PROPERTY PUBLIC Busy : BOOL
GET
Busy := asyncResponse <> 0;
END_GET
END_PROPERTY

METHOD PUBLIC CyclicCall
VAR_INPUT
END_VAR
timer(in := Busy, pt := T#1S);

IF timer.Q THEN
	asyncResponse.CompleteWithString(result);
	asyncResponse := 0;
	result := '';
END_IF
END_METHOD

METHOD Handle
VAR_INPUT
	Parameters : I_Deserializer;
	Response : I_SynchronousRpcResponse;
END_VAR
VAR
	deserializerFeedback : DeserializerFeedback;
	echo : T_MAXSTRING;
END_VAR
IF Busy THEN
	Response.RejectWithError('HANDLER_TOO_BUSY','Already processing response');
	RETURN;
END_IF

IF NOT Parameters.TryGetKeyString('Echo', echo, deserializerFeedback) THEN
	Response.RejectWithError('MISSING_PARAMETER','Missing Echo parameter');
	RETURN;
END_IF

result := echo;
Response.TryMakeAsynchronous(asyncResponse);
END_METHOD

END_FUNCTION_BLOCK

// ---- mobject-server/Mocks/RejectWithMessageAsyncHandler.TcPOU
FUNCTION_BLOCK RejectWithMessageAsyncHandler IMPLEMENTS I_AsynchronousRpcHandler
VAR
END_VAR

METHOD Handle
VAR_INPUT
	Parameters : I_Deserializer;
	Response : I_AsynchronousRpcResponse;
END_VAR
VAR
END_VAR
Response.RejectWithError('EXAMPLE_ERROR_CODE','This is the reject message');
END_METHOD

END_FUNCTION_BLOCK

// ---- mobject-server/Mocks/RejectWithMessageSyncHandler.TcPOU
FUNCTION_BLOCK RejectWithMessageSyncHandler IMPLEMENTS I_SynchronousRpcHandler
VAR
END_VAR

METHOD Handle
VAR_INPUT
	Parameters : I_Deserializer;
	Response : I_SynchronousRpcResponse;
END_VAR
VAR
END_VAR
Response.RejectWithError('EXAMPLE_ERROR_CODE','This is the reject message');
END_METHOD

END_FUNCTION_BLOCK

// ---- mobject-server/_Internal/ChunkedRequestData_TestSuite.TcPOU
FUNCTION_BLOCK ChunkedRequestData_TestSuite EXTENDS TcUnit.FB_TestSuite
VAR
END_VAR

TestChunkedPayloadStoredCorrectly_10Chunks();
TestChunkedPayloadStoredCorrectly_2Chunks();
TestCorrectPayloadSizeInBytes_20Bytes();
TestCorrectPayloadSizeInBytes_100Bytes();
TestIsCompleteOnceAllChunksAdded();
TestTryAddChunkedPayloadReturnsFalseWhenTooBig();
TestTryAddChunkedPayloadReturnsTrueWhenValid();
TestTryAddChunkedPayloadRejectsOutOfOrderChunk();
TestTryAddChunkedPayloadRejectsDuplicateChunk();

METHOD TestChunkedPayloadStoredCorrectly_10Chunks
VAR
	chunkedRequestData : ChunkedRequestData(3,10); // results in 30 bytes
	dataChunk1 : STRING(2) := 'ab'; // results in 3 bytes
	dataChunk2 : STRING(2) := 'cd'; // results in 3 bytes
	dataChunk3 : STRING(2) := 'ef'; // results in 3 bytes
	dataChunk4 : STRING(2) := 'gh'; // results in 3 bytes
	dataChunk5 : STRING(2) := 'ij'; // results in 3 bytes
	dataChunk6 : STRING(2) := 'kl'; // results in 3 bytes
	dataChunk7 : STRING(2) := 'mn'; // results in 3 bytes
	dataChunk8 : STRING(2) := 'op'; // results in 3 bytes
	dataChunk9 : STRING(2) := 'qr'; // results in 3 bytes
	dataChunk10 : STRING(2) := 'st'; // results in 3 bytes
	dataAddress : PVOID;
	dataSize : UDINT;
	result : STRING(29);
	expected : STRING(29) := 'abcdefghijklmnopqrst'; // results in 30 bytes
END_VAR
TEST('TestChunkedPayloadStoredCorrectly_10Chunks');

memset(ADR(result),0,SIZEOF(result));

chunkedRequestData.TryAddChunkedPayload(ADR(dataChunk1), SIZEOF(dataChunk1), 1);
chunkedRequestData.TryAddChunkedPayload(ADR(dataChunk2), SIZEOF(dataChunk2), 2);
chunkedRequestData.TryAddChunkedPayload(ADR(dataChunk3), SIZEOF(dataChunk3), 3);
chunkedRequestData.TryAddChunkedPayload(ADR(dataChunk4), SIZEOF(dataChunk4), 4);
chunkedRequestData.TryAddChunkedPayload(ADR(dataChunk5), SIZEOF(dataChunk5), 5);
chunkedRequestData.TryAddChunkedPayload(ADR(dataChunk6), SIZEOF(dataChunk6), 6);
chunkedRequestData.TryAddChunkedPayload(ADR(dataChunk7), SIZEOF(dataChunk7), 7);
chunkedRequestData.TryAddChunkedPayload(ADR(dataChunk8), SIZEOF(dataChunk8), 8);
chunkedRequestData.TryAddChunkedPayload(ADR(dataChunk9), SIZEOF(dataChunk9), 9);
chunkedRequestData.TryAddChunkedPayload(ADR(dataChunk10), SIZEOF(dataChunk10), 10);

dataAddress := chunkedRequestData.PayloadAddress;
dataSize := chunkedRequestData.PayloadSizeInBytes;

memcpy(ADR(result),dataAddress,dataSize);

AssertEquals(
	Expected := expected,
	Actual := result,
	Message := 'Did not correctly assemble the chunked string data'
);

TEST_FINISHED();
END_METHOD

METHOD TestChunkedPayloadStoredCorrectly_2Chunks
VAR
	chunkedRequestData : ChunkedRequestData(4,2); // results in 8 bytes
	dataChunk1 : STRING(3) := 'foo'; // results in 4 bytes
	dataChunk2 : STRING(3) := 'bar'; // results in 4 bytes
	dataAddress : PVOID;
	dataSize : UDINT;
	result : STRING(7);
	expected : STRING(7) := 'foobar'; // results in 8 bytes
END_VAR
TEST('TestChunkedPayloadStoredCorrectly_2Chunks');

memset(ADR(result),0,SIZEOF(result));

chunkedRequestData.TryAddChunkedPayload(ADR(dataChunk1), SIZEOF(dataChunk1), 1);
chunkedRequestData.TryAddChunkedPayload(ADR(dataChunk2), SIZEOF(dataChunk2), 2);

dataAddress := chunkedRequestData.PayloadAddress;
dataSize := chunkedRequestData.PayloadSizeInBytes;

memcpy(ADR(result),dataAddress,dataSize);

AssertEquals(
	Expected := expected,
	Actual := result,
	Message := 'Did not correctly assemble the chunked string data'
);

TEST_FINISHED();
END_METHOD

METHOD TestCorrectPayloadSizeInBytes_100Bytes
VAR
	chunkedRequestData : ChunkedRequestData(20,5);
	result : UDINT;
	expected : UDINT := 100;
END_VAR
TEST('TestCorrectPayloadSizeInBytes_100Bytes');

result := chunkedRequestData.PayloadSizeInBytes;

AssertEquals(
	Expected := expected,
	Actual := result,
	Message := 'Did not create the correct payload size based on the constructor arguments'
);

TEST_FINISHED();
END_METHOD

METHOD TestCorrectPayloadSizeInBytes_20Bytes
VAR
	chunkedRequestData : ChunkedRequestData(2,10);
	result : UDINT;
	expected : UDINT := 20;
END_VAR
TEST('TestCorrectPayloadSizeInBytes_20Bytes');

result := chunkedRequestData.PayloadSizeInBytes;

AssertEquals(
	Expected := expected,
	Actual := result,
	Message := 'Did not create the correct payload size based on the constructor arguments'
);

TEST_FINISHED();
END_METHOD

METHOD TestIsCompleteOnceAllChunksAdded
VAR
	chunkedRequestData : ChunkedRequestData(4,2);
	dataChunk1 : STRING(3) := 'foo';
	dataChunk2 : STRING(3) := 'bar';
	isComplete : BOOL;
END_VAR
TEST('TestIsCompleteOnceAllChunksAdded');

isComplete := chunkedRequestData.IsComplete;

AssertFalse(
	Condition := isComplete,
	Message := 'Incorrectly reported as IsComplete with 0/2 chunks added'
);

chunkedRequestData.TryAddChunkedPayload(ADR(dataChunk1), SIZEOF(dataChunk1), 1);
isComplete := chunkedRequestData.IsComplete;

AssertFalse(
	Condition := isComplete,
	Message := 'Incorrectly reported as IsComplete with 1/2 chunks added'
);

chunkedRequestData.TryAddChunkedPayload(ADR(dataChunk2), SIZEOF(dataChunk2), 2);
isComplete := chunkedRequestData.IsComplete;

AssertTrue(
	Condition := isComplete,
	Message := 'Failed to reported IsComplete with 2/2 chunks added'
);

TEST_FINISHED();
END_METHOD

METHOD TestTryAddChunkedPayloadReturnsFalseWhenTooBig
VAR
	chunkedRequestData : ChunkedRequestData(4,1);
	dataChunk : STRING(10) := 'foo';
	added : BOOL;
END_VAR
TEST('TestTryAddChunkedPayloadReturnsFalseWhenTooBig');

added := chunkedRequestData.TryAddChunkedPayload(ADR(dataChunk), SIZEOF(dataChunk), 1);

AssertFalse(
	Condition := added,
	Message := 'Incorrectly reported that the try was successful'
);

TEST_FINISHED();
END_METHOD

METHOD TestTryAddChunkedPayloadRejectsOutOfOrderChunk
VAR
	chunkedRequestData : ChunkedRequestData(4,3);
	dataChunk : STRING(3) := 'foo';
	added : BOOL;
END_VAR
TEST('TestTryAddChunkedPayloadRejectsOutOfOrderChunk');

// chunk 2 arriving before chunk 1 cannot be appended in the right place
added := chunkedRequestData.TryAddChunkedPayload(ADR(dataChunk), SIZEOF(dataChunk), 2);

AssertFalse(
	Condition := added,
	Message := 'A chunk which is not the one due next must be rejected, not appended out of order'
);

TEST_FINISHED();
END_METHOD

METHOD TestTryAddChunkedPayloadRejectsDuplicateChunk
VAR
	chunkedRequestData : ChunkedRequestData(4,3);
	dataChunk : STRING(3) := 'foo';
	firstAdd : BOOL;
	duplicateAdd : BOOL;
END_VAR
TEST('TestTryAddChunkedPayloadRejectsDuplicateChunk');

firstAdd := chunkedRequestData.TryAddChunkedPayload(ADR(dataChunk), SIZEOF(dataChunk), 1);
duplicateAdd := chunkedRequestData.TryAddChunkedPayload(ADR(dataChunk), SIZEOF(dataChunk), 1);

AssertTrue(
	Condition := firstAdd,
	Message := 'The first chunk should have been accepted'
);

// resending chunk 1 would otherwise append it twice and count twice towards completion
AssertFalse(
	Condition := duplicateAdd,
	Message := 'A repeated chunk must be rejected rather than appended a second time'
);

TEST_FINISHED();
END_METHOD

METHOD TestTryAddChunkedPayloadReturnsTrueWhenValid
VAR
	chunkedRequestData : ChunkedRequestData(4,1);
	dataChunk : STRING(3) := 'foo';
	added : BOOL;
END_VAR
TEST('TestTryAddChunkedPayloadReturnsTrueWhenValid');

added := chunkedRequestData.TryAddChunkedPayload(ADR(dataChunk), SIZEOF(dataChunk), 1);

AssertTrue(
	Condition := added,
	Message := 'Incorrectly reported that the try failed'
);

TEST_FINISHED();
END_METHOD

END_FUNCTION_BLOCK

// ---- mobject-server/_Internal/AsyncResponseSessionData_TestSuite.TcPOU
FUNCTION_BLOCK AsyncResponseSessionData_TestSuite EXTENDS TcUnit.FB_TestSuite
VAR
END_VAR

TestNewResponseIsPending();
TestFreshResponseHasNotExpired();
TestZeroMaxAgeDisablesTheDeadline();
TestCompletedResponseIsNoLongerPending();
TestRejectedResponseIsNoLongerPending();

METHOD TestCompletedResponseIsNoLongerPending
VAR
	asyncResponseSessionData : AsyncResponseSessionData(SuggestedRetryDelayInMs := 0, MaxAge := T#60S);
END_VAR
TEST('TestCompletedResponseIsNoLongerPending');

asyncResponseSessionData.Success();

AssertFalse(
	Condition := asyncResponseSessionData.IsPending,
	Message := 'A response which has completed should no longer report as pending'
);

TEST_FINISHED();
END_METHOD

METHOD TestFreshResponseHasNotExpired
VAR
	asyncResponseSessionData : AsyncResponseSessionData(SuggestedRetryDelayInMs := 0, MaxAge := T#60S);
END_VAR
TEST('TestFreshResponseHasNotExpired');

AssertFalse(
	Condition := asyncResponseSessionData.HasExpired,
	Message := 'A response created this cycle cannot already be past a 60s deadline'
);

TEST_FINISHED();
END_METHOD

METHOD TestNewResponseIsPending
VAR
	asyncResponseSessionData : AsyncResponseSessionData(SuggestedRetryDelayInMs := 0, MaxAge := T#60S);
END_VAR
TEST('TestNewResponseIsPending');

AssertTrue(
	Condition := asyncResponseSessionData.IsPending,
	Message := 'A newly created response should be pending until the handler completes it'
);

TEST_FINISHED();
END_METHOD

METHOD TestRejectedResponseIsNoLongerPending
VAR
	asyncResponseSessionData : AsyncResponseSessionData(SuggestedRetryDelayInMs := 0, MaxAge := T#60S);
END_VAR
TEST('TestRejectedResponseIsNoLongerPending');

asyncResponseSessionData.Error('SOME_CODE', 'some message');

AssertFalse(
	Condition := asyncResponseSessionData.IsPending,
	Message := 'A response which has been rejected should no longer report as pending'
);

TEST_FINISHED();
END_METHOD

METHOD TestZeroMaxAgeDisablesTheDeadline
VAR
	asyncResponseSessionData : AsyncResponseSessionData(SuggestedRetryDelayInMs := 0, MaxAge := T#0S);
END_VAR
TEST('TestZeroMaxAgeDisablesTheDeadline');

// T#0S is the documented way to switch the deadline off.  It must not be read
// as 'expires immediately', which would fail every asynchronous call.
AssertFalse(
	Condition := asyncResponseSessionData.HasExpired,
	Message := 'A max age of T#0S should disable the deadline, not expire instantly'
);

TEST_FINISHED();
END_METHOD

END_FUNCTION_BLOCK

// ---- mobject-server/Mocks/AdjustableSizeReplyRpcHandler.TcPOU
FUNCTION_BLOCK AdjustableSizeReplyRpcHandler IMPLEMENTS I_SynchronousRpcHandler
VAR
END_VAR

METHOD Handle
VAR_INPUT
	Parameters : I_Deserializer;
	Response : I_SynchronousRpcResponse;
END_VAR
VAR
	deserializerFeedback : DeserializerFeedback;
	size : UDINT;
	pBytes : POINTER TO BYTE;
	currentPos : POINTER TO BYTE;
	i : UDINT;
	count : BYTE;
END_VAR
IF NOT Parameters.TryGetKeyUdint('Size', size, deserializerFeedback) THEN
	Response.RejectWithError('MISSING_PARAMETER','Missing Size parameter');
	RETURN;
END_IF

IF size = 0 THEN 
	Response.CompleteWithNull();
END_IF

pBytes := __NEW(BYTE, size);
FOR i := 0 TO size -1 DO
	currentPos := pBytes + i;
	currentPos^ := count;
	count := count + 1;
END_FOR

Response.CompleteWithBytesAsHex(pBytes, UDINT_TO_DINT(size));

__Delete(pBytes);
END_METHOD

END_FUNCTION_BLOCK

// ---- mobject-collections/MobjectCollectionsExample.TcPOU
PROGRAM MobjectCollectionsExample
VAR
END_VAR

END_PROGRAM

// ---- mobject-collections/Tests/Mocks/EventHandlers/CollectionEventHandlerBase.TcPOU
FUNCTION_BLOCK ABSTRACT CollectionEventHandlerBase IMPLEMENTS I_EventHandler
VAR
	_eventReceived : BOOL;
	fromExpected : BOOL;
END_VAR

PROPERTY PUBLIC EventReceived : BOOL
GET // PUBLIC
EventReceived := _eventReceived;
END_GET
END_PROPERTY

PROPERTY PUBLIC FromExpectedOriginator : BOOL
GET // PUBLIC
FromExpectedOriginator := fromExpected;
END_GET
END_PROPERTY

METHOD PUBLIC ABSTRACT HandleEvent
VAR_INPUT
	Event : I_Event;
END_VAR
END_METHOD

METHOD PUBLIC Reset
_eventReceived := FALSE;
fromExpected := FALSE;
END_METHOD

END_FUNCTION_BLOCK

// ---- mobject-collections/Tests/Mocks/EventHandlers/KeyValueCollectionDisposedEventHandler.TcPOU
FUNCTION_BLOCK KeyValueCollectionDisposedEventHandler EXTENDS KeyValueCollectionEventHandler

METHOD PUBLIC HandleEvent
VAR_INPUT
	Event : I_Event;
END_VAR
VAR
	disposedEvent : I_KeyValueCollectionDisposedEvent;
END_VAR
IF __QUERYINTERFACE(Event, disposedEvent) THEN
	_eventReceived := TRUE;
	fromExpected := disposedEvent.Target = expectedOriginator;
END_IF
END_METHOD

END_FUNCTION_BLOCK

// ---- mobject-collections/Tests/Mocks/EventHandlers/KeyValueCollectionEventHandler.TcPOU
FUNCTION_BLOCK ABSTRACT KeyValueCollectionEventHandler EXTENDS CollectionEventHandlerBase
VAR
	expectedOriginator : I_KeyValueCollection;
END_VAR

METHOD FB_init : BOOL
VAR_INPUT
	bInitRetains : BOOL; // if TRUE, the retain variables are initialized (warm start / cold start)
	bInCopyCode : BOOL;  // if TRUE, the instance afterwards gets moved into the copy code (online change)
	ExpectedOriginator : I_KeyValueCollection;
END_VAR
SetExpectedOriginator(ExpectedOriginator);
END_METHOD

METHOD PUBLIC SetExpectedOriginator
VAR_INPUT
	ExpectedOriginator : I_KeyValueCollection;
END_VAR
THIS^.expectedOriginator := ExpectedOriginator;
END_METHOD

END_FUNCTION_BLOCK

// ---- mobject-converters/Tests/BYTE_TO_TestSuite.TcPOU
FUNCTION_BLOCK PUBLIC BYTE_TO_TestSuite EXTENDS TcUnit.FB_TestSuite
VAR
END_VAR

Check_BYTE_TO_BOOL_Max();
Check_BYTE_TO_BOOL_Min();
Check_BYTE_TO_BYTE_Max();
Check_BYTE_TO_BYTE_Min();
Check_BYTE_TO_WORD_Max();
Check_BYTE_TO_WORD_Min();
Check_BYTE_TO_DWORD_Max();
Check_BYTE_TO_DWORD_Min();
Check_BYTE_TO_LWORD_Max();
Check_BYTE_TO_LWORD_Min();
Check_BYTE_TO_SINT_Max();
Check_BYTE_TO_SINT_Min();
Check_BYTE_TO_SINT_TooHigh();
Check_BYTE_TO_INT_Max();
Check_BYTE_TO_INT_Min();
Check_BYTE_TO_DINT_Max();
Check_BYTE_TO_DINT_Min();
Check_BYTE_TO_LINT_Max();
Check_BYTE_TO_LINT_Min();
Check_BYTE_TO_USINT_Max();
Check_BYTE_TO_USINT_Min();
Check_BYTE_TO_UINT_Max();
Check_BYTE_TO_UINT_Min();
Check_BYTE_TO_UDINT_Max();
Check_BYTE_TO_UDINT_Min();
Check_BYTE_TO_ULINT_Max();
Check_BYTE_TO_ULINT_Min();
Check_BYTE_TO_REAL_Max();
Check_BYTE_TO_REAL_Min();
Check_BYTE_TO_LREAL_Max();
Check_BYTE_TO_LREAL_Min();
Check_BYTE_TO_TIME_Max();
Check_BYTE_TO_TIME_Min();
Check_BYTE_TO_TOD_Max();
Check_BYTE_TO_TOD_Min();
Check_BYTE_TO_DATE_Max();
Check_BYTE_TO_DATE_Min();
Check_BYTE_TO_DT_Max();
Check_BYTE_TO_DT_Min();
Check_BYTE_TO_STRING_Max();
Check_BYTE_TO_STRING_Min();

METHOD PUBLIC Check_BYTE_TO_BOOL_Max
VAR
	value : BYTE := DatatypeLimits.BYTE_MAX_VALUE;
	actual : BOOL;
	converted : BOOL;
	equal : BOOL;
END_VAR
TEST('Check_BYTE_TO_BOOL_Max');

// @TEST-RUN
converted := TryConvert_BYTE_TO_Destination(value, actual);
equal := actual = BYTE_TO_BOOL(value);

// @TEST-ASSERT
AssertTrue(Condition := equal, Message := 'Did not convert BYTE to BOOL correctly');
AssertTrue(Condition := converted, Message := 'Did not report BYTE to BOOL conversion was successful');

TEST_FINISHED();
END_METHOD

METHOD PUBLIC Check_BYTE_TO_BOOL_Min
VAR
	value : BYTE := DatatypeLimits.BYTE_MIN_VALUE;
	actual : BOOL;
	converted : BOOL;
	equal : BOOL;
END_VAR
TEST('Check_BYTE_TO_BOOL_Min');

// @TEST-RUN
converted := TryConvert_BYTE_TO_Destination(value, actual);
equal := actual = BYTE_TO_BOOL(value);

// @TEST-ASSERT
AssertTrue(Condition := equal, Message := 'Did not convert BYTE to BOOL correctly');
AssertTrue(Condition := converted, Message := 'Did not report BYTE to BOOL conversion was successful');

TEST_FINISHED();
END_METHOD

METHOD PUBLIC Check_BYTE_TO_BYTE_Max
VAR
	value : BYTE := DatatypeLimits.BYTE_MAX_VALUE;
	actual : BYTE;
	converted : BOOL;
	equal : BOOL;
END_VAR
TEST('Check_BYTE_TO_BYTE_Max');

// @TEST-RUN
converted := TryConvert_BYTE_TO_Destination(value, actual);
equal := actual = value;

// @TEST-ASSERT
AssertTrue(Condition := equal, Message := 'Did not convert BYTE to BYTE correctly');
AssertTrue(Condition := converted, Message := 'Did not report BYTE to BYTE conversion was successful');

TEST_FINISHED();
END_METHOD

METHOD PUBLIC Check_BYTE_TO_BYTE_Min
VAR
	value : BYTE := DatatypeLimits.BYTE_MIN_VALUE;
	actual : BYTE;
	converted : BOOL;
	equal : BOOL;
END_VAR
TEST('Check_BYTE_TO_BYTE_Min');

// @TEST-RUN
converted := TryConvert_BYTE_TO_Destination(value, actual);
equal := actual = value;

// @TEST-ASSERT
AssertTrue(Condition := equal, Message := 'Did not convert BYTE to BYTE correctly');
AssertTrue(Condition := converted, Message := 'Did not report BYTE to BYTE conversion was successful');

TEST_FINISHED();
END_METHOD

METHOD PUBLIC Check_BYTE_TO_DATE_Max
VAR
	value : BYTE := DatatypeLimits.BYTE_MAX_VALUE;
	actual : DATE;
	converted : BOOL;
	equal : BOOL;
END_VAR
TEST('Check_BYTE_TO_DATE_Max');

// @TEST-RUN
converted := TryConvert_BYTE_TO_Destination(value, actual);
equal := actual = BYTE_TO_DATE(value);

// @TEST-ASSERT
AssertTrue(Condition := equal, Message := 'Did not convert BYTE to DATE correctly');
AssertTrue(Condition := converted, Message := 'Did not report BYTE to DATE conversion was successful');

TEST_FINISHED();
END_METHOD

METHOD PUBLIC Check_BYTE_TO_DATE_Min
VAR
	value : BYTE := DatatypeLimits.BYTE_MIN_VALUE;
	actual : DATE;
	converted : BOOL;
	equal : BOOL;
END_VAR
TEST('Check_BYTE_TO_DATE_Min');

// @TEST-RUN
converted := TryConvert_BYTE_TO_Destination(value, actual);
equal := actual = BYTE_TO_DATE(value);

// @TEST-ASSERT
AssertTrue(Condition := equal, Message := 'Did not convert BYTE to DATE correctly');
AssertTrue(Condition := converted, Message := 'Did not report BYTE to DATE conversion was successful');

TEST_FINISHED();
END_METHOD

METHOD PUBLIC Check_BYTE_TO_DINT_Max
VAR
	value : BYTE := DatatypeLimits.BYTE_MAX_VALUE;
	actual : DINT;
	converted : BOOL;
	equal : BOOL;
END_VAR
TEST('Check_BYTE_TO_DINT_Max');

// @TEST-RUN
converted := TryConvert_BYTE_TO_Destination(value, actual);
equal := actual = BYTE_TO_DINT(value);

// @TEST-ASSERT
AssertTrue(Condition := equal, Message := 'Did not convert BYTE to DINT correctly');
AssertTrue(Condition := converted, Message := 'Did not report BYTE to DINT conversion was successful');

TEST_FINISHED();
END_METHOD

METHOD PUBLIC Check_BYTE_TO_DINT_Min
VAR
	value : BYTE := DatatypeLimits.BYTE_MIN_VALUE;
	actual : DINT;
	converted : BOOL;
	equal : BOOL;
END_VAR
TEST('Check_BYTE_TO_DINT_Min');

// @TEST-RUN
converted := TryConvert_BYTE_TO_Destination(value, actual);
equal := actual = BYTE_TO_DINT(value);

// @TEST-ASSERT
AssertTrue(Condition := equal, Message := 'Did not convert BYTE to DINT correctly');
AssertTrue(Condition := converted, Message := 'Did not report BYTE to DINT conversion was successful');

TEST_FINISHED();
END_METHOD

METHOD PUBLIC Check_BYTE_TO_DT_Max
VAR
	value : BYTE := DatatypeLimits.BYTE_MAX_VALUE;
	actual : DT;
	converted : BOOL;
	equal : BOOL;
END_VAR
TEST('Check_BYTE_TO_DT_Max');

// @TEST-RUN
converted := TryConvert_BYTE_TO_Destination(value, actual);
equal := actual = BYTE_TO_DT(value);

// @TEST-ASSERT
AssertTrue(Condition := equal, Message := 'Did not convert BYTE to DT correctly');
AssertTrue(Condition := converted, Message := 'Did not report BYTE to DT conversion was successful');

TEST_FINISHED();
END_METHOD

METHOD PUBLIC Check_BYTE_TO_DT_Min
VAR
	value : BYTE := DatatypeLimits.BYTE_MIN_VALUE;
	actual : DT;
	converted : BOOL;
	equal : BOOL;
END_VAR
TEST('Check_BYTE_TO_DT_Min');

// @TEST-RUN
converted := TryConvert_BYTE_TO_Destination(value, actual);
equal := actual = BYTE_TO_DT(value);

// @TEST-ASSERT
AssertTrue(Condition := equal, Message := 'Did not convert BYTE to DT correctly');
AssertTrue(Condition := converted, Message := 'Did not report BYTE to DT conversion was successful');

TEST_FINISHED();
END_METHOD

METHOD PUBLIC Check_BYTE_TO_DWORD_Max
VAR
	value : BYTE := DatatypeLimits.BYTE_MAX_VALUE;
	actual : DWORD;
	converted : BOOL;
	equal : BOOL;
END_VAR
TEST('Check_BYTE_TO_DWORD_Max');

// @TEST-RUN
converted := TryConvert_BYTE_TO_Destination(value, actual);
equal := actual = BYTE_TO_DWORD(value);

// @TEST-ASSERT
AssertTrue(Condition := equal, Message := 'Did not convert BYTE to DWORD correctly');
AssertTrue(Condition := converted, Message := 'Did not report BYTE to DWORD conversion was successful');

TEST_FINISHED();
END_METHOD

METHOD PUBLIC Check_BYTE_TO_DWORD_Min
VAR
	value : BYTE := DatatypeLimits.BYTE_MIN_VALUE;
	actual : DWORD;
	converted : BOOL;
	equal : BOOL;
END_VAR
TEST('Check_BYTE_TO_DWORD_Min');

// @TEST-RUN
converted := TryConvert_BYTE_TO_Destination(value, actual);
equal := actual = BYTE_TO_DWORD(value);

// @TEST-ASSERT
AssertTrue(Condition := equal, Message := 'Did not convert BYTE to DWORD correctly');
AssertTrue(Condition := converted, Message := 'Did not report BYTE to DWORD conversion was successful');

TEST_FINISHED();
END_METHOD

METHOD PUBLIC Check_BYTE_TO_INT_Max
VAR
	value : BYTE := DatatypeLimits.BYTE_MAX_VALUE;
	actual : INT;
	converted : BOOL;
	equal : BOOL;
END_VAR
TEST('Check_BYTE_TO_INT_Max');

// @TEST-RUN
converted := TryConvert_BYTE_TO_Destination(value, actual);
equal := actual = BYTE_TO_INT(value);

// @TEST-ASSERT
AssertTrue(Condition := equal, Message := 'Did not convert BYTE to INT correctly');
AssertTrue(Condition := converted, Message := 'Did not report BYTE to INT conversion was successful');

TEST_FINISHED();
END_METHOD

METHOD PUBLIC Check_BYTE_TO_INT_Min
VAR
	value : BYTE := DatatypeLimits.BYTE_MIN_VALUE;
	actual : INT;
	converted : BOOL;
	equal : BOOL;
END_VAR
TEST('Check_BYTE_TO_INT_Min');

// @TEST-RUN
converted := TryConvert_BYTE_TO_Destination(value, actual);
equal := actual = BYTE_TO_INT(value);

// @TEST-ASSERT
AssertTrue(Condition := equal, Message := 'Did not convert BYTE to INT correctly');
AssertTrue(Condition := converted, Message := 'Did not report BYTE to INT conversion was successful');

TEST_FINISHED();
END_METHOD

METHOD PUBLIC Check_BYTE_TO_LINT_Max
VAR
	value : BYTE := DatatypeLimits.BYTE_MAX_VALUE;
	actual : LINT;
	converted : BOOL;
	equal : BOOL;
END_VAR
TEST('Check_BYTE_TO_LINT_Max');

// @TEST-RUN
converted := TryConvert_BYTE_TO_Destination(value, actual);
equal := actual = BYTE_TO_LINT(value);

// @TEST-ASSERT
AssertTrue(Condition := equal, Message := 'Did not convert BYTE to LINT correctly');
AssertTrue(Condition := converted, Message := 'Did not report BYTE to LINT conversion was successful');

TEST_FINISHED();
END_METHOD

METHOD PUBLIC Check_BYTE_TO_LINT_Min
VAR
	value : BYTE := DatatypeLimits.BYTE_MIN_VALUE;
	actual : LINT;
	converted : BOOL;
	equal : BOOL;
END_VAR
TEST('Check_BYTE_TO_LINT_Min');

// @TEST-RUN
converted := TryConvert_BYTE_TO_Destination(value, actual);
equal := actual = BYTE_TO_LINT(value);

// @TEST-ASSERT
AssertTrue(Condition := equal, Message := 'Did not convert BYTE to LINT correctly');
AssertTrue(Condition := converted, Message := 'Did not report BYTE to LINT conversion was successful');

TEST_FINISHED();
END_METHOD

METHOD PUBLIC Check_BYTE_TO_LREAL_Max
VAR
	value : BYTE := DatatypeLimits.BYTE_MAX_VALUE;
	actual : LREAL;
	converted : BOOL;
	equal : BOOL;
END_VAR
TEST('Check_BYTE_TO_LREAL_Max');

// @TEST-RUN
converted := TryConvert_BYTE_TO_Destination(value, actual);
equal := actual = BYTE_TO_LREAL(value);

// @TEST-ASSERT
AssertTrue(Condition := equal, Message := 'Did not convert BYTE to LREAL correctly');
AssertTrue(Condition := converted, Message := 'Did not report BYTE to LREAL conversion was successful');

TEST_FINISHED();
END_METHOD

METHOD PUBLIC Check_BYTE_TO_LREAL_Min
VAR
	value : BYTE := DatatypeLimits.BYTE_MIN_VALUE;
	actual : LREAL;
	converted : BOOL;
	equal : BOOL;
END_VAR
TEST('Check_BYTE_TO_LREAL_Min');

// @TEST-RUN
converted := TryConvert_BYTE_TO_Destination(value, actual);
equal := actual = BYTE_TO_LREAL(value);

// @TEST-ASSERT
AssertTrue(Condition := equal, Message := 'Did not convert BYTE to LREAL correctly');
AssertTrue(Condition := converted, Message := 'Did not report BYTE to LREAL conversion was successful');

TEST_FINISHED();
END_METHOD

METHOD PUBLIC Check_BYTE_TO_LWORD_Max
VAR
	value : BYTE := DatatypeLimits.BYTE_MAX_VALUE;
	actual : LWORD;
	converted : BOOL;
	equal : BOOL;
END_VAR
TEST('Check_BYTE_TO_LWORD_Max');

// @TEST-RUN
converted := TryConvert_BYTE_TO_Destination(value, actual);
equal := actual = BYTE_TO_LWORD(value);

// @TEST-ASSERT
AssertTrue(Condition := equal, Message := 'Did not convert BYTE to LWORD correctly');
AssertTrue(Condition := converted, Message := 'Did not report BYTE to LWORD conversion was successful');

TEST_FINISHED();
END_METHOD

METHOD PUBLIC Check_BYTE_TO_LWORD_Min
VAR
	value : BYTE := DatatypeLimits.BYTE_MIN_VALUE;
	actual : LWORD;
	converted : BOOL;
	equal : BOOL;
END_VAR
TEST('Check_BYTE_TO_LWORD_Min');

// @TEST-RUN
converted := TryConvert_BYTE_TO_Destination(value, actual);
equal := actual = BYTE_TO_LWORD(value);

// @TEST-ASSERT
AssertTrue(Condition := equal, Message := 'Did not convert BYTE to LWORD correctly');
AssertTrue(Condition := converted, Message := 'Did not report BYTE to LWORD conversion was successful');

TEST_FINISHED();
END_METHOD

METHOD PUBLIC Check_BYTE_TO_REAL_Max
VAR
	value : BYTE := DatatypeLimits.BYTE_MAX_VALUE;
	actual : REAL;
	converted : BOOL;
	equal : BOOL;
END_VAR
TEST('Check_BYTE_TO_REAL_Max');

// @TEST-RUN
converted := TryConvert_BYTE_TO_Destination(value, actual);
equal := actual = BYTE_TO_REAL(value);

// @TEST-ASSERT
AssertTrue(Condition := equal, Message := 'Did not convert BYTE to REAL correctly');
AssertTrue(Condition := converted, Message := 'Did not report BYTE to REAL conversion was successful');

TEST_FINISHED();
END_METHOD

METHOD PUBLIC Check_BYTE_TO_REAL_Min
VAR
	value : BYTE := DatatypeLimits.BYTE_MIN_VALUE;
	actual : REAL;
	converted : BOOL;
	equal : BOOL;
END_VAR
TEST('Check_BYTE_TO_REAL_Min');

// @TEST-RUN
converted := TryConvert_BYTE_TO_Destination(value, actual);
equal := actual = BYTE_TO_REAL(value);

// @TEST-ASSERT
AssertTrue(Condition := equal, Message := 'Did not convert BYTE to REAL correctly');
AssertTrue(Condition := converted, Message := 'Did not report BYTE to REAL conversion was successful');

TEST_FINISHED();
END_METHOD

METHOD PUBLIC Check_BYTE_TO_SINT_Max
VAR
	value : BYTE := DatatypeLimits.MAX_VALUE_OF_BYTE_WHICH_CAN_BE_HELD_IN_A_SINT;
	actual : SINT;
	converted : BOOL;
	equal : BOOL;
END_VAR
TEST('Check_BYTE_TO_SINT_Max');

// @TEST-RUN
converted := TryConvert_BYTE_TO_Destination(value, actual);
equal := actual = BYTE_TO_SINT(value);

// @TEST-ASSERT
AssertTrue(Condition := equal, Message := 'Did not convert BYTE to SINT correctly');
AssertTrue(Condition := converted, Message := 'Did not report BYTE to SINT conversion was successful');

TEST_FINISHED();
END_METHOD

METHOD PUBLIC Check_BYTE_TO_SINT_Min
VAR
	value : BYTE := DatatypeLimits.BYTE_MIN_VALUE;
	actual : SINT;
	converted : BOOL;
	equal : BOOL;
END_VAR
TEST('Check_BYTE_TO_SINT_Min');

// @TEST-RUN
converted := TryConvert_BYTE_TO_Destination(value, actual);
equal := actual = BYTE_TO_SINT(value);

// @TEST-ASSERT
AssertTrue(Condition := equal, Message := 'Did not convert BYTE to SINT correctly');
AssertTrue(Condition := converted, Message := 'Did not report BYTE to SINT conversion was successful');

TEST_FINISHED();
END_METHOD

METHOD PUBLIC Check_BYTE_TO_SINT_TooHigh
VAR
	value : BYTE := DatatypeLimits.BYTE_MAX_VALUE;
	actual : SINT;
	converted : BOOL;
END_VAR
TEST('Check_BYTE_TO_SINT_TooHigh');

// @TEST-RUN
converted := TryConvert_BYTE_TO_Destination(value, actual);

// @TEST-ASSERT
AssertFalse(Condition := converted, Message := 'Did not report BYTE to SINT conversion was prevented');

TEST_FINISHED();
END_METHOD

METHOD PUBLIC Check_BYTE_TO_STRING_Max
VAR
	value : BYTE := DatatypeLimits.BYTE_MAX_VALUE;
	actual : STRING;
	converted : BOOL;
	equal : BOOL;
END_VAR
TEST('Check_BYTE_TO_STRING_Max');

// @TEST-RUN
converted := TryConvert_BYTE_TO_Destination(value, actual);
equal := actual = BYTE_TO_STRING(value);

// @TEST-ASSERT
AssertTrue(Condition := equal, Message := 'Did not convert BYTE to STRING correctly');
AssertTrue(Condition := converted, Message := 'Did not report BYTE to STRING conversion was successful');

TEST_FINISHED();
END_METHOD

METHOD PUBLIC Check_BYTE_TO_STRING_Min
VAR
	value : BYTE := DatatypeLimits.BYTE_MIN_VALUE;
	actual : STRING;
	converted : BOOL;
	equal : BOOL;
END_VAR
TEST('Check_BYTE_TO_STRING_Min');

// @TEST-RUN
converted := TryConvert_BYTE_TO_Destination(value, actual);
equal := actual = BYTE_TO_STRING(value);

// @TEST-ASSERT
AssertTrue(Condition := equal, Message := 'Did not convert BYTE to STRING correctly');
AssertTrue(Condition := converted, Message := 'Did not report BYTE to STRING conversion was successful');

TEST_FINISHED();
END_METHOD

METHOD PUBLIC Check_BYTE_TO_TIME_Max
VAR
	value : BYTE := DatatypeLimits.BYTE_MAX_VALUE;
	actual : TIME;
	converted : BOOL;
	equal : BOOL;
END_VAR
TEST('Check_BYTE_TO_TIME_Max');

// @TEST-RUN
converted := TryConvert_BYTE_TO_Destination(value, actual);
equal := actual = BYTE_TO_TIME(value);

// @TEST-ASSERT
AssertTrue(Condition := equal, Message := 'Did not convert BYTE to TIME correctly');
AssertTrue(Condition := converted, Message := 'Did not report BYTE to TIME conversion was successful');

TEST_FINISHED();
END_METHOD

METHOD PUBLIC Check_BYTE_TO_TIME_Min
VAR
	value : BYTE := DatatypeLimits.BYTE_MIN_VALUE;
	actual : TIME;
	converted : BOOL;
	equal : BOOL;
END_VAR
TEST('Check_BYTE_TO_TIME_Min');

// @TEST-RUN
converted := TryConvert_BYTE_TO_Destination(value, actual);
equal := actual = BYTE_TO_TIME(value);

// @TEST-ASSERT
AssertTrue(Condition := equal, Message := 'Did not convert BYTE to TIME correctly');
AssertTrue(Condition := converted, Message := 'Did not report BYTE to TIME conversion was successful');

TEST_FINISHED();
END_METHOD

METHOD PUBLIC Check_BYTE_TO_TOD_Max
VAR
	value : BYTE := DatatypeLimits.BYTE_MAX_VALUE;
	actual : TOD;
	converted : BOOL;
	equal : BOOL;
END_VAR
TEST('Check_BYTE_TO_TOD_Max');

// @TEST-RUN
converted := TryConvert_BYTE_TO_Destination(value, actual);
equal := actual = BYTE_TO_TOD(value);

// @TEST-ASSERT
AssertTrue(Condition := equal, Message := 'Did not convert BYTE to TOD correctly');
AssertTrue(Condition := converted, Message := 'Did not report BYTE to TOD conversion was successful');

TEST_FINISHED();
END_METHOD

METHOD PUBLIC Check_BYTE_TO_TOD_Min
VAR
	value : BYTE := DatatypeLimits.BYTE_MIN_VALUE;
	actual : TOD;
	converted : BOOL;
	equal : BOOL;
END_VAR
TEST('Check_BYTE_TO_TOD_Min');

// @TEST-RUN
converted := TryConvert_BYTE_TO_Destination(value, actual);
equal := actual = BYTE_TO_TOD(value);

// @TEST-ASSERT
AssertTrue(Condition := equal, Message := 'Did not convert BYTE to TOD correctly');
AssertTrue(Condition := converted, Message := 'Did not report BYTE to TOD conversion was successful');

TEST_FINISHED();
END_METHOD

METHOD PUBLIC Check_BYTE_TO_UDINT_Max
VAR
	value : BYTE := DatatypeLimits.BYTE_MAX_VALUE;
	actual : UDINT;
	converted : BOOL;
	equal : BOOL;
END_VAR
TEST('Check_BYTE_TO_UDINT_Max');

// @TEST-RUN
converted := TryConvert_BYTE_TO_Destination(value, actual);
equal := actual = BYTE_TO_UDINT(value);

// @TEST-ASSERT
AssertTrue(Condition := equal, Message := 'Did not convert BYTE to UDINT correctly');
AssertTrue(Condition := converted, Message := 'Did not report BYTE to UDINT conversion was successful');

TEST_FINISHED();
END_METHOD

METHOD PUBLIC Check_BYTE_TO_UDINT_Min
VAR
	value : BYTE := DatatypeLimits.BYTE_MIN_VALUE;
	actual : UDINT;
	converted : BOOL;
	equal : BOOL;
END_VAR
TEST('Check_BYTE_TO_UDINT_Min');

// @TEST-RUN
converted := TryConvert_BYTE_TO_Destination(value, actual);
equal := actual = BYTE_TO_UDINT(value);

// @TEST-ASSERT
AssertTrue(Condition := equal, Message := 'Did not convert BYTE to UDINT correctly');
AssertTrue(Condition := converted, Message := 'Did not report BYTE to UDINT conversion was successful');

TEST_FINISHED();
END_METHOD

METHOD PUBLIC Check_BYTE_TO_UINT_Max
VAR
	value : BYTE := DatatypeLimits.BYTE_MAX_VALUE;
	actual : UINT;
	converted : BOOL;
	equal : BOOL;
END_VAR
TEST('Check_BYTE_TO_UINT_Max');

// @TEST-RUN
converted := TryConvert_BYTE_TO_Destination(value, actual);
equal := actual = BYTE_TO_UINT(value);

// @TEST-ASSERT
AssertTrue(Condition := equal, Message := 'Did not convert BYTE to UINT correctly');
AssertTrue(Condition := converted, Message := 'Did not report BYTE to UINT conversion was successful');

TEST_FINISHED();
END_METHOD

METHOD PUBLIC Check_BYTE_TO_UINT_Min
VAR
	value : BYTE := DatatypeLimits.BYTE_MIN_VALUE;
	actual : UINT;
	converted : BOOL;
	equal : BOOL;
END_VAR
TEST('Check_BYTE_TO_UINT_Min');

// @TEST-RUN
converted := TryConvert_BYTE_TO_Destination(value, actual);
equal := actual = BYTE_TO_UINT(value);

// @TEST-ASSERT
AssertTrue(Condition := equal, Message := 'Did not convert BYTE to UINT correctly');
AssertTrue(Condition := converted, Message := 'Did not report BYTE to UINT conversion was successful');

TEST_FINISHED();
END_METHOD

METHOD PUBLIC Check_BYTE_TO_ULINT_Max
VAR
	value : BYTE := DatatypeLimits.BYTE_MAX_VALUE;
	actual : ULINT;
	converted : BOOL;
	equal : BOOL;
END_VAR
TEST('Check_BYTE_TO_ULINT_Max');

// @TEST-RUN
converted := TryConvert_BYTE_TO_Destination(value, actual);
equal := actual = BYTE_TO_ULINT(value);

// @TEST-ASSERT
AssertTrue(Condition := equal, Message := 'Did not convert BYTE to ULINT correctly');
AssertTrue(Condition := converted, Message := 'Did not report BYTE to ULINT conversion was successful');

TEST_FINISHED();
END_METHOD

METHOD PUBLIC Check_BYTE_TO_ULINT_Min
VAR
	value : BYTE := DatatypeLimits.BYTE_MIN_VALUE;
	actual : ULINT;
	converted : BOOL;
	equal : BOOL;
END_VAR
TEST('Check_BYTE_TO_ULINT_Min');

// @TEST-RUN
converted := TryConvert_BYTE_TO_Destination(value, actual);
equal := actual = BYTE_TO_ULINT(value);

// @TEST-ASSERT
AssertTrue(Condition := equal, Message := 'Did not convert BYTE to ULINT correctly');
AssertTrue(Condition := converted, Message := 'Did not report BYTE to ULINT conversion was successful');

TEST_FINISHED();
END_METHOD

METHOD PUBLIC Check_BYTE_TO_USINT_Max
VAR
	value : BYTE := DatatypeLimits.BYTE_MAX_VALUE;
	actual : USINT;
	converted : BOOL;
	equal : BOOL;
END_VAR
TEST('Check_BYTE_TO_USINT_Max');

// @TEST-RUN
converted := TryConvert_BYTE_TO_Destination(value, actual);
equal := actual = BYTE_TO_USINT(value);

// @TEST-ASSERT
AssertTrue(Condition := equal, Message := 'Did not convert BYTE to USINT correctly');
AssertTrue(Condition := converted, Message := 'Did not report BYTE to USINT conversion was successful');

TEST_FINISHED();
END_METHOD

METHOD PUBLIC Check_BYTE_TO_USINT_Min
VAR
	value : BYTE := DatatypeLimits.BYTE_MIN_VALUE;
	actual : USINT;
	converted : BOOL;
	equal : BOOL;
END_VAR
TEST('Check_BYTE_TO_USINT_Min');

// @TEST-RUN
converted := TryConvert_BYTE_TO_Destination(value, actual);
equal := actual = BYTE_TO_USINT(value);

// @TEST-ASSERT
AssertTrue(Condition := equal, Message := 'Did not convert BYTE to USINT correctly');
AssertTrue(Condition := converted, Message := 'Did not report BYTE to USINT conversion was successful');

TEST_FINISHED();
END_METHOD

METHOD PUBLIC Check_BYTE_TO_WORD_Max
VAR
	value : BYTE := DatatypeLimits.BYTE_MAX_VALUE;
	actual : WORD;
	converted : BOOL;
	equal : BOOL;
END_VAR
TEST('Check_BYTE_TO_WORD_Max');

// @TEST-RUN
converted := TryConvert_BYTE_TO_Destination(value, actual);
equal := actual = BYTE_TO_WORD(value);

// @TEST-ASSERT
AssertTrue(Condition := equal, Message := 'Did not convert BYTE to WORD correctly');
AssertTrue(Condition := converted, Message := 'Did not report BYTE to WORD conversion was successful');

TEST_FINISHED();
END_METHOD

METHOD PUBLIC Check_BYTE_TO_WORD_Min
VAR
	value : BYTE := DatatypeLimits.BYTE_MIN_VALUE;
	actual : WORD;
	converted : BOOL;
	equal : BOOL;
END_VAR
TEST('Check_BYTE_TO_WORD_Min');

// @TEST-RUN
converted := TryConvert_BYTE_TO_Destination(value, actual);
equal := actual = BYTE_TO_WORD(value);

// @TEST-ASSERT
AssertTrue(Condition := equal, Message := 'Did not convert BYTE to WORD correctly');
AssertTrue(Condition := converted, Message := 'Did not report BYTE to WORD conversion was successful');

TEST_FINISHED();
END_METHOD

END_FUNCTION_BLOCK

// ---- mobject-converters/Tests/DATE_TO_TestSuite.TcPOU
FUNCTION_BLOCK PUBLIC DATE_TO_TestSuite EXTENDS TcUnit.FB_TestSuite
VAR
END_VAR

Check_DATE_TO_BOOL_Max();
Check_DATE_TO_BOOL_Min();
Check_DATE_TO_BYTE_Max();
Check_DATE_TO_BYTE_Min();
Check_DATE_TO_BYTE_TooHigh();
Check_DATE_TO_WORD_Max();
Check_DATE_TO_WORD_Min();
Check_DATE_TO_WORD_TooHigh();
Check_DATE_TO_DWORD_Max();
Check_DATE_TO_DWORD_Min();
Check_DATE_TO_LWORD_Max();
Check_DATE_TO_LWORD_Min();
Check_DATE_TO_SINT_Max();
Check_DATE_TO_SINT_Min();
Check_DATE_TO_SINT_TooHigh();
Check_DATE_TO_INT_Max();
Check_DATE_TO_INT_Min();
Check_DATE_TO_INT_TooHigh();
Check_DATE_TO_DINT_Max();
Check_DATE_TO_DINT_Min();
Check_DATE_TO_DINT_TooHigh();
Check_DATE_TO_LINT_Max();
Check_DATE_TO_LINT_Min();
Check_DATE_TO_USINT_Max();
Check_DATE_TO_USINT_Min();
Check_DATE_TO_USINT_TooHigh();
Check_DATE_TO_UINT_Max();
Check_DATE_TO_UINT_Min();
Check_DATE_TO_UINT_TooHigh();
Check_DATE_TO_UDINT_Max();
Check_DATE_TO_UDINT_Min();
Check_DATE_TO_ULINT_Max();
Check_DATE_TO_ULINT_Min();
Check_DATE_TO_REAL_Max();
Check_DATE_TO_REAL_Min();
Check_DATE_TO_LREAL_Max();
Check_DATE_TO_LREAL_Min();
Check_DATE_TO_TIME_Max();
Check_DATE_TO_TIME_Min();
Check_DATE_TO_TIME_TooHigh();
Check_DATE_TO_TOD_Max();
Check_DATE_TO_TOD_Min();
Check_DATE_TO_TOD_TooHigh();
Check_DATE_TO_DATE_Max();
Check_DATE_TO_DATE_Min();
Check_DATE_TO_DT_Max();
Check_DATE_TO_DT_Min();
Check_DATE_TO_STRING_Max();
Check_DATE_TO_STRING_Min();

METHOD PUBLIC Check_DATE_TO_BOOL_Max
VAR
	value : DATE := DatatypeLimits.DATE_MAX_VALUE;
	actual : BOOL;
	converted : BOOL;
	equal : BOOL;
END_VAR
TEST('Check_DATE_TO_BOOL_Max');

// @TEST-RUN
converted := TryConvert_DATE_TO_Destination(value, actual);
equal := actual = DATE_TO_BOOL(value);

// @TEST-ASSERT
AssertTrue(Condition := equal, Message := 'Did not convert DATE to BOOL correctly');
AssertTrue(Condition := converted, Message := 'Did not report DATE to BOOL conversion was successful');

TEST_FINISHED();
END_METHOD

METHOD PUBLIC Check_DATE_TO_BOOL_Min
VAR
	value : DATE := DatatypeLimits.DATE_MIN_VALUE;
	actual : BOOL;
	converted : BOOL;
	equal : BOOL;
END_VAR
TEST('Check_DATE_TO_BOOL_Min');

// @TEST-RUN
converted := TryConvert_DATE_TO_Destination(value, actual);
equal := actual = DATE_TO_BOOL(value);

// @TEST-ASSERT
AssertTrue(Condition := equal, Message := 'Did not convert DATE to BOOL correctly');
AssertTrue(Condition := converted, Message := 'Did not report DATE to BOOL conversion was successful');

TEST_FINISHED();
END_METHOD

METHOD PUBLIC Check_DATE_TO_BYTE_Max
VAR
	value : DATE := DatatypeLimits.MAX_VALUE_OF_DATE_WHICH_CAN_BE_HELD_IN_A_BYTE;
	actual : BYTE;
	converted : BOOL;
	equal : BOOL;
END_VAR
TEST('Check_DATE_TO_BYTE_Max');

// @TEST-RUN
converted := TryConvert_DATE_TO_Destination(value, actual);
equal := actual = DATE_TO_BYTE(value);

// @TEST-ASSERT
AssertTrue(Condition := equal, Message := 'Did not convert DATE to BYTE correctly');
AssertTrue(Condition := converted, Message := 'Did not report DATE to BYTE conversion was successful');

TEST_FINISHED();
END_METHOD

METHOD PUBLIC Check_DATE_TO_BYTE_Min
VAR
	value : DATE := DatatypeLimits.DATE_MIN_VALUE;
	actual : BYTE;
	converted : BOOL;
	equal : BOOL;
END_VAR
TEST('Check_DATE_TO_BYTE_Min');

// @TEST-RUN
converted := TryConvert_DATE_TO_Destination(value, actual);
equal := actual = DATE_TO_BYTE(value);

// @TEST-ASSERT
AssertTrue(Condition := equal, Message := 'Did not convert DATE to BYTE correctly');
AssertTrue(Condition := converted, Message := 'Did not report DATE to BYTE conversion was successful');

TEST_FINISHED();
END_METHOD

METHOD PUBLIC Check_DATE_TO_BYTE_TooHigh
VAR
	value : DATE := DatatypeLimits.DATE_MAX_VALUE;
	actual : BYTE;
	converted : BOOL;
END_VAR
TEST('Check_DATE_TO_BYTE_TooHigh');

// @TEST-RUN
converted := TryConvert_DATE_TO_Destination(value, actual);

// @TEST-ASSERT
AssertFalse(Condition := converted, Message := 'Did not report DATE to BYTE conversion was prevented');

TEST_FINISHED();
END_METHOD

METHOD PUBLIC Check_DATE_TO_DATE_Max
VAR
	value : DATE := DatatypeLimits.DATE_MAX_VALUE;
	actual : DATE;
	converted : BOOL;
	equal : BOOL;
END_VAR
TEST('Check_DATE_TO_DATE_Max');

// @TEST-RUN
converted := TryConvert_DATE_TO_Destination(value, actual);
equal := actual = value;

// @TEST-ASSERT
AssertTrue(Condition := equal, Message := 'Did not convert DATE to DATE correctly');
AssertTrue(Condition := converted, Message := 'Did not report DATE to DATE conversion was successful');

TEST_FINISHED();
END_METHOD

METHOD PUBLIC Check_DATE_TO_DATE_Min
VAR
	value : DATE := DatatypeLimits.DATE_MIN_VALUE;
	actual : DATE;
	converted : BOOL;
	equal : BOOL;
END_VAR
TEST('Check_DATE_TO_DATE_Min');

// @TEST-RUN
converted := TryConvert_DATE_TO_Destination(value, actual);
equal := actual = value;

// @TEST-ASSERT
AssertTrue(Condition := equal, Message := 'Did not convert DATE to DATE correctly');
AssertTrue(Condition := converted, Message := 'Did not report DATE to DATE conversion was successful');

TEST_FINISHED();
END_METHOD

METHOD PUBLIC Check_DATE_TO_DINT_Max
VAR
	value : DATE := DatatypeLimits.MAX_VALUE_OF_DATE_WHICH_CAN_BE_HELD_IN_A_DINT;
	actual : DINT;
	converted : BOOL;
	equal : BOOL;
END_VAR
TEST('Check_DATE_TO_DINT_Max');

// @TEST-RUN
converted := TryConvert_DATE_TO_Destination(value, actual);
equal := actual = DATE_TO_DINT(value);

// @TEST-ASSERT
AssertTrue(Condition := equal, Message := 'Did not convert DATE to DINT correctly');
AssertTrue(Condition := converted, Message := 'Did not report DATE to DINT conversion was successful');

TEST_FINISHED();
END_METHOD

METHOD PUBLIC Check_DATE_TO_DINT_Min
VAR
	value : DATE := DatatypeLimits.DATE_MIN_VALUE;
	actual : DINT;
	converted : BOOL;
	equal : BOOL;
END_VAR
TEST('Check_DATE_TO_DINT_Min');

// @TEST-RUN
converted := TryConvert_DATE_TO_Destination(value, actual);
equal := actual = DATE_TO_DINT(value);

// @TEST-ASSERT
AssertTrue(Condition := equal, Message := 'Did not convert DATE to DINT correctly');
AssertTrue(Condition := converted, Message := 'Did not report DATE to DINT conversion was successful');

TEST_FINISHED();
END_METHOD

METHOD PUBLIC Check_DATE_TO_DINT_TooHigh
VAR
	value : DATE := DatatypeLimits.DATE_MAX_VALUE;
	actual : DINT;
	converted : BOOL;
END_VAR
TEST('Check_DATE_TO_DINT_TooHigh');

// @TEST-RUN
converted := TryConvert_DATE_TO_Destination(value, actual);

// @TEST-ASSERT
AssertFalse(Condition := converted, Message := 'Did not report DATE to DINT conversion was prevented');

TEST_FINISHED();
END_METHOD

METHOD PUBLIC Check_DATE_TO_DT_Max
VAR
	value : DATE := DatatypeLimits.MAX_VALUE_OF_DATE_WHICH_CAN_BE_HELD_IN_A_DT;
	actual : DT;
	converted : BOOL;
	equal : BOOL;
END_VAR
TEST('Check_DATE_TO_DT_Max');

// @TEST-RUN
converted := TryConvert_DATE_TO_Destination(value, actual);
equal := actual = DATE_TO_DT(value);

// @TEST-ASSERT
AssertTrue(Condition := equal, Message := 'Did not convert DATE to DT correctly');
AssertTrue(Condition := converted, Message := 'Did not report DATE to DT conversion was successful');

TEST_FINISHED();
END_METHOD

METHOD PUBLIC Check_DATE_TO_DT_Min
VAR
	value : DATE := DatatypeLimits.DATE_MIN_VALUE;
	actual : DT;
	converted : BOOL;
	equal : BOOL;
END_VAR
TEST('Check_DATE_TO_DT_Min');

// @TEST-RUN
converted := TryConvert_DATE_TO_Destination(value, actual);
equal := actual = DATE_TO_DT(value);

// @TEST-ASSERT
AssertTrue(Condition := equal, Message := 'Did not convert DATE to DT correctly');
AssertTrue(Condition := converted, Message := 'Did not report DATE to DT conversion was successful');

TEST_FINISHED();
END_METHOD

METHOD PUBLIC Check_DATE_TO_DWORD_Max
VAR
	value : DATE := DatatypeLimits.DATE_MAX_VALUE;
	actual : DWORD;
	converted : BOOL;
	equal : BOOL;
END_VAR
TEST('Check_DATE_TO_DWORD_Max');

// @TEST-RUN
converted := TryConvert_DATE_TO_Destination(value, actual);
equal := actual = DATE_TO_DWORD(value);

// @TEST-ASSERT
AssertTrue(Condition := equal, Message := 'Did not convert DATE to DWORD correctly');
AssertTrue(Condition := converted, Message := 'Did not report DATE to DWORD conversion was successful');

TEST_FINISHED();
END_METHOD

METHOD PUBLIC Check_DATE_TO_DWORD_Min
VAR
	value : DATE := DatatypeLimits.DATE_MIN_VALUE;
	actual : DWORD;
	converted : BOOL;
	equal : BOOL;
END_VAR
TEST('Check_DATE_TO_DWORD_Min');

// @TEST-RUN
converted := TryConvert_DATE_TO_Destination(value, actual);
equal := actual = DATE_TO_DWORD(value);

// @TEST-ASSERT
AssertTrue(Condition := equal, Message := 'Did not convert DATE to DWORD correctly');
AssertTrue(Condition := converted, Message := 'Did not report DATE to DWORD conversion was successful');

TEST_FINISHED();
END_METHOD

METHOD PUBLIC Check_DATE_TO_INT_Max
VAR
	value : DATE := DatatypeLimits.MAX_VALUE_OF_DATE_WHICH_CAN_BE_HELD_IN_A_INT;
	actual : INT;
	converted : BOOL;
	equal : BOOL;
END_VAR
TEST('Check_DATE_TO_INT_Max');

// @TEST-RUN
converted := TryConvert_DATE_TO_Destination(value, actual);
equal := actual = DATE_TO_INT(value);

// @TEST-ASSERT
AssertTrue(Condition := equal, Message := 'Did not convert DATE to INT correctly');
AssertTrue(Condition := converted, Message := 'Did not report DATE to INT conversion was successful');

TEST_FINISHED();
END_METHOD

METHOD PUBLIC Check_DATE_TO_INT_Min
VAR
	value : DATE := DatatypeLimits.DATE_MIN_VALUE;
	actual : INT;
	converted : BOOL;
	equal : BOOL;
END_VAR
TEST('Check_DATE_TO_INT_Min');

// @TEST-RUN
converted := TryConvert_DATE_TO_Destination(value, actual);
equal := actual = DATE_TO_INT(value);

// @TEST-ASSERT
AssertTrue(Condition := equal, Message := 'Did not convert DATE to INT correctly');
AssertTrue(Condition := converted, Message := 'Did not report DATE to INT conversion was successful');

TEST_FINISHED();
END_METHOD

METHOD PUBLIC Check_DATE_TO_INT_TooHigh
VAR
	value : DATE := DatatypeLimits.DATE_MAX_VALUE;
	actual : INT;
	converted : BOOL;
END_VAR
TEST('Check_DATE_TO_INT_TooHigh');

// @TEST-RUN
converted := TryConvert_DATE_TO_Destination(value, actual);

// @TEST-ASSERT
AssertFalse(Condition := converted, Message := 'Did not report DATE to INT conversion was prevented');

TEST_FINISHED();
END_METHOD

METHOD PUBLIC Check_DATE_TO_LINT_Max
VAR
	value : DATE := DatatypeLimits.DATE_MAX_VALUE;
	actual : LINT;
	converted : BOOL;
	equal : BOOL;
END_VAR
TEST('Check_DATE_TO_LINT_Max');

// @TEST-RUN
converted := TryConvert_DATE_TO_Destination(value, actual);
equal := actual = DATE_TO_LINT(value);

// @TEST-ASSERT
AssertTrue(Condition := equal, Message := 'Did not convert DATE to LINT correctly');
AssertTrue(Condition := converted, Message := 'Did not report DATE to LINT conversion was successful');

TEST_FINISHED();
END_METHOD

METHOD PUBLIC Check_DATE_TO_LINT_Min
VAR
	value : DATE := DatatypeLimits.DATE_MIN_VALUE;
	actual : LINT;
	converted : BOOL;
	equal : BOOL;
END_VAR
TEST('Check_DATE_TO_LINT_Min');

// @TEST-RUN
converted := TryConvert_DATE_TO_Destination(value, actual);
equal := actual = DATE_TO_LINT(value);

// @TEST-ASSERT
AssertTrue(Condition := equal, Message := 'Did not convert DATE to LINT correctly');
AssertTrue(Condition := converted, Message := 'Did not report DATE to LINT conversion was successful');

TEST_FINISHED();
END_METHOD

METHOD PUBLIC Check_DATE_TO_LREAL_Max
VAR
	value : DATE := DatatypeLimits.DATE_MAX_VALUE;
	actual : LREAL;
	converted : BOOL;
	equal : BOOL;
END_VAR
TEST('Check_DATE_TO_LREAL_Max');

// @TEST-RUN
converted := TryConvert_DATE_TO_Destination(value, actual);
equal := actual = DATE_TO_LREAL(value);

// @TEST-ASSERT
AssertTrue(Condition := equal, Message := 'Did not convert DATE to LREAL correctly');
AssertTrue(Condition := converted, Message := 'Did not report DATE to LREAL conversion was successful');

TEST_FINISHED();
END_METHOD

METHOD PUBLIC Check_DATE_TO_LREAL_Min
VAR
	value : DATE := DatatypeLimits.DATE_MIN_VALUE;
	actual : LREAL;
	converted : BOOL;
	equal : BOOL;
END_VAR
TEST('Check_DATE_TO_LREAL_Min');

// @TEST-RUN
converted := TryConvert_DATE_TO_Destination(value, actual);
equal := actual = DATE_TO_LREAL(value);

// @TEST-ASSERT
AssertTrue(Condition := equal, Message := 'Did not convert DATE to LREAL correctly');
AssertTrue(Condition := converted, Message := 'Did not report DATE to LREAL conversion was successful');

TEST_FINISHED();
END_METHOD

METHOD PUBLIC Check_DATE_TO_LWORD_Max
VAR
	value : DATE := DatatypeLimits.DATE_MAX_VALUE;
	actual : LWORD;
	converted : BOOL;
	equal : BOOL;
END_VAR
TEST('Check_DATE_TO_LWORD_Max');

// @TEST-RUN
converted := TryConvert_DATE_TO_Destination(value, actual);
equal := actual = DATE_TO_LWORD(value);

// @TEST-ASSERT
AssertTrue(Condition := equal, Message := 'Did not convert DATE to LWORD correctly');
AssertTrue(Condition := converted, Message := 'Did not report DATE to LWORD conversion was successful');

TEST_FINISHED();
END_METHOD

METHOD PUBLIC Check_DATE_TO_LWORD_Min
VAR
	value : DATE := DatatypeLimits.DATE_MIN_VALUE;
	actual : LWORD;
	converted : BOOL;
	equal : BOOL;
END_VAR
TEST('Check_DATE_TO_LWORD_Min');

// @TEST-RUN
converted := TryConvert_DATE_TO_Destination(value, actual);
equal := actual = DATE_TO_LWORD(value);

// @TEST-ASSERT
AssertTrue(Condition := equal, Message := 'Did not convert DATE to LWORD correctly');
AssertTrue(Condition := converted, Message := 'Did not report DATE to LWORD conversion was successful');

TEST_FINISHED();
END_METHOD

METHOD PUBLIC Check_DATE_TO_REAL_Max
VAR
	value : DATE := DatatypeLimits.DATE_MAX_VALUE;
	actual : REAL;
	converted : BOOL;
	equal : BOOL;
END_VAR
TEST('Check_DATE_TO_REAL_Max');

// @TEST-RUN
converted := TryConvert_DATE_TO_Destination(value, actual);
equal := actual = DATE_TO_REAL(value);

// @TEST-ASSERT
AssertTrue(Condition := equal, Message := 'Did not convert DATE to REAL correctly');
AssertTrue(Condition := converted, Message := 'Did not report DATE to REAL conversion was successful');

TEST_FINISHED();
END_METHOD

METHOD PUBLIC Check_DATE_TO_REAL_Min
VAR
	value : DATE := DatatypeLimits.DATE_MIN_VALUE;
	actual : REAL;
	converted : BOOL;
	equal : BOOL;
END_VAR
TEST('Check_DATE_TO_REAL_Min');

// @TEST-RUN
converted := TryConvert_DATE_TO_Destination(value, actual);
equal := actual = DATE_TO_REAL(value);

// @TEST-ASSERT
AssertTrue(Condition := equal, Message := 'Did not convert DATE to REAL correctly');
AssertTrue(Condition := converted, Message := 'Did not report DATE to REAL conversion was successful');

TEST_FINISHED();
END_METHOD

METHOD PUBLIC Check_DATE_TO_SINT_Max
VAR
	value : DATE := DatatypeLimits.MAX_VALUE_OF_DATE_WHICH_CAN_BE_HELD_IN_A_SINT;
	actual : SINT;
	converted : BOOL;
	equal : BOOL;
END_VAR
TEST('Check_DATE_TO_SINT_Max');

// @TEST-RUN
converted := TryConvert_DATE_TO_Destination(value, actual);
equal := actual = DATE_TO_SINT(value);

// @TEST-ASSERT
AssertTrue(Condition := equal, Message := 'Did not convert DATE to SINT correctly');
AssertTrue(Condition := converted, Message := 'Did not report DATE to SINT conversion was successful');

TEST_FINISHED();
END_METHOD

METHOD PUBLIC Check_DATE_TO_SINT_Min
VAR
	value : DATE := DatatypeLimits.DATE_MIN_VALUE;
	actual : SINT;
	converted : BOOL;
	equal : BOOL;
END_VAR
TEST('Check_DATE_TO_SINT_Min');

// @TEST-RUN
converted := TryConvert_DATE_TO_Destination(value, actual);
equal := actual = DATE_TO_SINT(value);

// @TEST-ASSERT
AssertTrue(Condition := equal, Message := 'Did not convert DATE to SINT correctly');
AssertTrue(Condition := converted, Message := 'Did not report DATE to SINT conversion was successful');

TEST_FINISHED();
END_METHOD

METHOD PUBLIC Check_DATE_TO_SINT_TooHigh
VAR
	value : DATE := DatatypeLimits.DATE_MAX_VALUE;
	actual : SINT;
	converted : BOOL;
END_VAR
TEST('Check_DATE_TO_SINT_TooHigh');

// @TEST-RUN
converted := TryConvert_DATE_TO_Destination(value, actual);

// @TEST-ASSERT
AssertFalse(Condition := converted, Message := 'Did not report DATE to SINT conversion was prevented');

TEST_FINISHED();
END_METHOD

METHOD PUBLIC Check_DATE_TO_STRING_Max
VAR
	value : DATE := DatatypeLimits.DATE_MAX_VALUE;
	actual : STRING;
	converted : BOOL;
	equal : BOOL;
END_VAR
TEST('Check_DATE_TO_STRING_Max');

// @TEST-RUN
converted := TryConvert_DATE_TO_Destination(value, actual);
equal := actual = DATE_TO_STRING(value);

// @TEST-ASSERT
AssertTrue(Condition := equal, Message := 'Did not convert DATE to STRING correctly');
AssertTrue(Condition := converted, Message := 'Did not report DATE to STRING conversion was successful');

TEST_FINISHED();
END_METHOD

METHOD PUBLIC Check_DATE_TO_STRING_Min
VAR
	value : DATE := DatatypeLimits.DATE_MIN_VALUE;
	actual : STRING;
	converted : BOOL;
	equal : BOOL;
END_VAR
TEST('Check_DATE_TO_STRING_Min');

// @TEST-RUN
converted := TryConvert_DATE_TO_Destination(value, actual);
equal := actual = DATE_TO_STRING(value);

// @TEST-ASSERT
AssertTrue(Condition := equal, Message := 'Did not convert DATE to STRING correctly');
AssertTrue(Condition := converted, Message := 'Did not report DATE to STRING conversion was successful');

TEST_FINISHED();
END_METHOD

METHOD PUBLIC Check_DATE_TO_TIME_Max
VAR
	value : DATE := DatatypeLimits.MAX_VALUE_OF_DATE_WHICH_CAN_BE_HELD_IN_A_TIME;
	actual : TIME;
	converted : BOOL;
	equal : BOOL;
END_VAR
TEST('Check_DATE_TO_TIME_Max');

// @TEST-RUN
converted := TryConvert_DATE_TO_Destination(value, actual);
equal := actual = DATE_TO_TIME(value);

// @TEST-ASSERT
AssertTrue(Condition := equal, Message := 'Did not convert DATE to TIME correctly');
AssertTrue(Condition := converted, Message := 'Did not report DATE to TIME conversion was successful');

TEST_FINISHED();
END_METHOD

METHOD PUBLIC Check_DATE_TO_TIME_Min
VAR
	value : DATE := DatatypeLimits.DATE_MIN_VALUE;
	actual : TIME;
	converted : BOOL;
	equal : BOOL;
END_VAR
TEST('Check_DATE_TO_TIME_Min');

// @TEST-RUN
converted := TryConvert_DATE_TO_Destination(value, actual);
equal := actual = DATE_TO_TIME(value);

// @TEST-ASSERT
AssertTrue(Condition := equal, Message := 'Did not convert DATE to TIME correctly');
AssertTrue(Condition := converted, Message := 'Did not report DATE to TIME conversion was successful');

TEST_FINISHED();
END_METHOD

METHOD PUBLIC Check_DATE_TO_TIME_TooHigh
VAR
	value : DATE := DatatypeLimits.DATE_MAX_VALUE;
	actual : TIME;
	converted : BOOL;
END_VAR
TEST('Check_DATE_TO_TIME_TooHigh');

// @TEST-RUN
converted := TryConvert_DATE_TO_Destination(value, actual);

// @TEST-ASSERT
AssertFalse(Condition := converted, Message := 'Did not report DATE to TIME conversion was prevented');

TEST_FINISHED();
END_METHOD

METHOD PUBLIC Check_DATE_TO_TOD_Max
VAR
	value : DATE := DatatypeLimits.MAX_VALUE_OF_DATE_WHICH_CAN_BE_HELD_IN_A_TOD;
	actual : TOD;
	converted : BOOL;
	equal : BOOL;
END_VAR
TEST('Check_DATE_TO_TOD_Max');

// @TEST-RUN
converted := TryConvert_DATE_TO_Destination(value, actual);
equal := actual = DATE_TO_TOD(value);

// @TEST-ASSERT
AssertTrue(Condition := equal, Message := 'Did not convert DATE to TOD correctly');
AssertTrue(Condition := converted, Message := 'Did not report DATE to TOD conversion was successful');

TEST_FINISHED();
END_METHOD

METHOD PUBLIC Check_DATE_TO_TOD_Min
VAR
	value : DATE := DatatypeLimits.DATE_MIN_VALUE;
	actual : TOD;
	converted : BOOL;
	equal : BOOL;
END_VAR
TEST('Check_DATE_TO_TOD_Min');

// @TEST-RUN
converted := TryConvert_DATE_TO_Destination(value, actual);
equal := actual = DATE_TO_TOD(value);

// @TEST-ASSERT
AssertTrue(Condition := equal, Message := 'Did not convert DATE to TOD correctly');
AssertTrue(Condition := converted, Message := 'Did not report DATE to TOD conversion was successful');

TEST_FINISHED();
END_METHOD

METHOD PUBLIC Check_DATE_TO_TOD_TooHigh
VAR
	value : DATE := DatatypeLimits.DATE_MAX_VALUE;
	actual : TOD;
	converted : BOOL;
END_VAR
TEST('Check_DATE_TO_TOD_TooHigh');

// @TEST-RUN
converted := TryConvert_DATE_TO_Destination(value, actual);

// @TEST-ASSERT
AssertFalse(Condition := converted, Message := 'Did not report DATE to TOD conversion was prevented');

TEST_FINISHED();
END_METHOD

METHOD PUBLIC Check_DATE_TO_UDINT_Max
VAR
	value : DATE := DatatypeLimits.DATE_MAX_VALUE;
	actual : UDINT;
	converted : BOOL;
	equal : BOOL;
END_VAR
TEST('Check_DATE_TO_UDINT_Max');

// @TEST-RUN
converted := TryConvert_DATE_TO_Destination(value, actual);
equal := actual = DATE_TO_UDINT(value);

// @TEST-ASSERT
AssertTrue(Condition := equal, Message := 'Did not convert DATE to UDINT correctly');
AssertTrue(Condition := converted, Message := 'Did not report DATE to UDINT conversion was successful');

TEST_FINISHED();
END_METHOD

METHOD PUBLIC Check_DATE_TO_UDINT_Min
VAR
	value : DATE := DatatypeLimits.DATE_MIN_VALUE;
	actual : UDINT;
	converted : BOOL;
	equal : BOOL;
END_VAR
TEST('Check_DATE_TO_UDINT_Min');

// @TEST-RUN
converted := TryConvert_DATE_TO_Destination(value, actual);
equal := actual = DATE_TO_UDINT(value);

// @TEST-ASSERT
AssertTrue(Condition := equal, Message := 'Did not convert DATE to UDINT correctly');
AssertTrue(Condition := converted, Message := 'Did not report DATE to UDINT conversion was successful');

TEST_FINISHED();
END_METHOD

METHOD PUBLIC Check_DATE_TO_UINT_Max
VAR
	value : DATE := DatatypeLimits.MAX_VALUE_OF_DATE_WHICH_CAN_BE_HELD_IN_A_UINT;
	actual : UINT;
	converted : BOOL;
	equal : BOOL;
END_VAR
TEST('Check_DATE_TO_UINT_Max');

// @TEST-RUN
converted := TryConvert_DATE_TO_Destination(value, actual);
equal := actual = DATE_TO_UINT(value);

// @TEST-ASSERT
AssertTrue(Condition := equal, Message := 'Did not convert DATE to UINT correctly');
AssertTrue(Condition := converted, Message := 'Did not report DATE to UINT conversion was successful');

TEST_FINISHED();
END_METHOD

METHOD PUBLIC Check_DATE_TO_UINT_Min
VAR
	value : DATE := DatatypeLimits.DATE_MIN_VALUE;
	actual : UINT;
	converted : BOOL;
	equal : BOOL;
END_VAR
TEST('Check_DATE_TO_UINT_Min');

// @TEST-RUN
converted := TryConvert_DATE_TO_Destination(value, actual);
equal := actual = DATE_TO_UINT(value);

// @TEST-ASSERT
AssertTrue(Condition := equal, Message := 'Did not convert DATE to UINT correctly');
AssertTrue(Condition := converted, Message := 'Did not report DATE to UINT conversion was successful');

TEST_FINISHED();
END_METHOD

METHOD PUBLIC Check_DATE_TO_UINT_TooHigh
VAR
	value : DATE := DatatypeLimits.DATE_MAX_VALUE;
	actual : UINT;
	converted : BOOL;
END_VAR
TEST('Check_DATE_TO_UINT_TooHigh');

// @TEST-RUN
converted := TryConvert_DATE_TO_Destination(value, actual);

// @TEST-ASSERT
AssertFalse(Condition := converted, Message := 'Did not report DATE to UINT conversion was prevented');

TEST_FINISHED();
END_METHOD

METHOD PUBLIC Check_DATE_TO_ULINT_Max
VAR
	value : DATE := DatatypeLimits.DATE_MAX_VALUE;
	actual : ULINT;
	converted : BOOL;
	equal : BOOL;
END_VAR
TEST('Check_DATE_TO_ULINT_Max');

// @TEST-RUN
converted := TryConvert_DATE_TO_Destination(value, actual);
equal := actual = DATE_TO_ULINT(value);

// @TEST-ASSERT
AssertTrue(Condition := equal, Message := 'Did not convert DATE to ULINT correctly');
AssertTrue(Condition := converted, Message := 'Did not report DATE to ULINT conversion was successful');

TEST_FINISHED();
END_METHOD

METHOD PUBLIC Check_DATE_TO_ULINT_Min
VAR
	value : DATE := DatatypeLimits.DATE_MIN_VALUE;
	actual : ULINT;
	converted : BOOL;
	equal : BOOL;
END_VAR
TEST('Check_DATE_TO_ULINT_Min');

// @TEST-RUN
converted := TryConvert_DATE_TO_Destination(value, actual);
equal := actual = DATE_TO_ULINT(value);

// @TEST-ASSERT
AssertTrue(Condition := equal, Message := 'Did not convert DATE to ULINT correctly');
AssertTrue(Condition := converted, Message := 'Did not report DATE to ULINT conversion was successful');

TEST_FINISHED();
END_METHOD

METHOD PUBLIC Check_DATE_TO_USINT_Max
VAR
	value : DATE := DatatypeLimits.MAX_VALUE_OF_DATE_WHICH_CAN_BE_HELD_IN_A_USINT;
	actual : USINT;
	converted : BOOL;
	equal : BOOL;
END_VAR
TEST('Check_DATE_TO_USINT_Max');

// @TEST-RUN
converted := TryConvert_DATE_TO_Destination(value, actual);
equal := actual = DATE_TO_USINT(value);

// @TEST-ASSERT
AssertTrue(Condition := equal, Message := 'Did not convert DATE to USINT correctly');
AssertTrue(Condition := converted, Message := 'Did not report DATE to USINT conversion was successful');

TEST_FINISHED();
END_METHOD

METHOD PUBLIC Check_DATE_TO_USINT_Min
VAR
	value : DATE := DatatypeLimits.DATE_MIN_VALUE;
	actual : USINT;
	converted : BOOL;
	equal : BOOL;
END_VAR
TEST('Check_DATE_TO_USINT_Min');

// @TEST-RUN
converted := TryConvert_DATE_TO_Destination(value, actual);
equal := actual = DATE_TO_USINT(value);

// @TEST-ASSERT
AssertTrue(Condition := equal, Message := 'Did not convert DATE to USINT correctly');
AssertTrue(Condition := converted, Message := 'Did not report DATE to USINT conversion was successful');

TEST_FINISHED();
END_METHOD

METHOD PUBLIC Check_DATE_TO_USINT_TooHigh
VAR
	value : DATE := DatatypeLimits.DATE_MAX_VALUE;
	actual : USINT;
	converted : BOOL;
END_VAR
TEST('Check_DATE_TO_USINT_TooHigh');

// @TEST-RUN
converted := TryConvert_DATE_TO_Destination(value, actual);

// @TEST-ASSERT
AssertFalse(Condition := converted, Message := 'Did not report DATE to USINT conversion was prevented');

TEST_FINISHED();
END_METHOD

METHOD PUBLIC Check_DATE_TO_WORD_Max
VAR
	value : DATE := DatatypeLimits.MAX_VALUE_OF_DATE_WHICH_CAN_BE_HELD_IN_A_WORD;
	actual : WORD;
	converted : BOOL;
	equal : BOOL;
END_VAR
TEST('Check_DATE_TO_WORD_Max');

// @TEST-RUN
converted := TryConvert_DATE_TO_Destination(value, actual);
equal := actual = DATE_TO_WORD(value);

// @TEST-ASSERT
AssertTrue(Condition := equal, Message := 'Did not convert DATE to WORD correctly');
AssertTrue(Condition := converted, Message := 'Did not report DATE to WORD conversion was successful');

TEST_FINISHED();
END_METHOD

METHOD PUBLIC Check_DATE_TO_WORD_Min
VAR
	value : DATE := DatatypeLimits.DATE_MIN_VALUE;
	actual : WORD;
	converted : BOOL;
	equal : BOOL;
END_VAR
TEST('Check_DATE_TO_WORD_Min');

// @TEST-RUN
converted := TryConvert_DATE_TO_Destination(value, actual);
equal := actual = DATE_TO_WORD(value);

// @TEST-ASSERT
AssertTrue(Condition := equal, Message := 'Did not convert DATE to WORD correctly');
AssertTrue(Condition := converted, Message := 'Did not report DATE to WORD conversion was successful');

TEST_FINISHED();
END_METHOD

METHOD PUBLIC Check_DATE_TO_WORD_TooHigh
VAR
	value : DATE := DatatypeLimits.DATE_MAX_VALUE;
	actual : WORD;
	converted : BOOL;
END_VAR
TEST('Check_DATE_TO_WORD_TooHigh');

// @TEST-RUN
converted := TryConvert_DATE_TO_Destination(value, actual);

// @TEST-ASSERT
AssertFalse(Condition := converted, Message := 'Did not report DATE to WORD conversion was prevented');

TEST_FINISHED();
END_METHOD

END_FUNCTION_BLOCK

// ---- mobject-converters/Tests/DINT_TO_TestSuite.TcPOU
FUNCTION_BLOCK PUBLIC DINT_TO_TestSuite EXTENDS TcUnit.FB_TestSuite
VAR
END_VAR

Check_DINT_TO_BOOL_Max();
Check_DINT_TO_BOOL_Min();
Check_DINT_TO_BYTE_Max();
Check_DINT_TO_BYTE_Min();
Check_DINT_TO_BYTE_TooHigh();
Check_DINT_TO_BYTE_TooLow();
Check_DINT_TO_WORD_Max();
Check_DINT_TO_WORD_Min();
Check_DINT_TO_WORD_TooHigh();
Check_DINT_TO_WORD_TooLow();
Check_DINT_TO_DWORD_Max();
Check_DINT_TO_DWORD_Min();
Check_DINT_TO_DWORD_TooLow();
Check_DINT_TO_LWORD_Max();
Check_DINT_TO_LWORD_Min();
Check_DINT_TO_LWORD_TooLow();
Check_DINT_TO_SINT_Max();
Check_DINT_TO_SINT_Min();
Check_DINT_TO_SINT_TooHigh();
Check_DINT_TO_SINT_TooLow();
Check_DINT_TO_INT_Max();
Check_DINT_TO_INT_Min();
Check_DINT_TO_INT_TooHigh();
Check_DINT_TO_INT_TooLow();
Check_DINT_TO_DINT_Max();
Check_DINT_TO_DINT_Min();
Check_DINT_TO_LINT_Max();
Check_DINT_TO_LINT_Min();
Check_DINT_TO_USINT_Max();
Check_DINT_TO_USINT_Min();
Check_DINT_TO_USINT_TooHigh();
Check_DINT_TO_USINT_TooLow();
Check_DINT_TO_UINT_Max();
Check_DINT_TO_UINT_Min();
Check_DINT_TO_UINT_TooHigh();
Check_DINT_TO_UINT_TooLow();
Check_DINT_TO_UDINT_Max();
Check_DINT_TO_UDINT_Min();
Check_DINT_TO_UDINT_TooLow();
Check_DINT_TO_ULINT_Max();
Check_DINT_TO_ULINT_Min();
Check_DINT_TO_ULINT_TooLow();
Check_DINT_TO_REAL_Max();
Check_DINT_TO_REAL_Min();
Check_DINT_TO_LREAL_Max();
Check_DINT_TO_LREAL_Min();
Check_DINT_TO_TIME_Max();
Check_DINT_TO_TIME_Min();
Check_DINT_TO_TIME_TooLow();
Check_DINT_TO_TOD_Max();
Check_DINT_TO_TOD_Min();
Check_DINT_TO_TOD_TooHigh();
Check_DINT_TO_TOD_TooLow();
Check_DINT_TO_DATE_Max();
Check_DINT_TO_DATE_Min();
Check_DINT_TO_DATE_TooLow();
Check_DINT_TO_DT_Max();
Check_DINT_TO_DT_Min();
Check_DINT_TO_DT_TooLow();
Check_DINT_TO_STRING_Max();
Check_DINT_TO_STRING_Min();

METHOD PUBLIC Check_DINT_TO_BOOL_Max
VAR
	value : DINT := DatatypeLimits.DINT_MAX_VALUE;
	actual : BOOL;
	converted : BOOL;
	equal : BOOL;
END_VAR
TEST('Check_DINT_TO_BOOL_Max');

// @TEST-RUN
converted := TryConvert_DINT_TO_Destination(value, actual);
equal := actual = DINT_TO_BOOL(value);

// @TEST-ASSERT
AssertTrue(Condition := equal, Message := 'Did not convert DINT to BOOL correctly');
AssertTrue(Condition := converted, Message := 'Did not report DINT to BOOL conversion was successful');

TEST_FINISHED();
END_METHOD

METHOD PUBLIC Check_DINT_TO_BOOL_Min
VAR
	value : DINT := DatatypeLimits.DINT_MIN_VALUE;
	actual : BOOL;
	converted : BOOL;
	equal : BOOL;
END_VAR
TEST('Check_DINT_TO_BOOL_Min');

// @TEST-RUN
converted := TryConvert_DINT_TO_Destination(value, actual);
equal := actual = DINT_TO_BOOL(value);

// @TEST-ASSERT
AssertTrue(Condition := equal, Message := 'Did not convert DINT to BOOL correctly');
AssertTrue(Condition := converted, Message := 'Did not report DINT to BOOL conversion was successful');

TEST_FINISHED();
END_METHOD

METHOD PUBLIC Check_DINT_TO_BYTE_Max
VAR
	value : DINT := DatatypeLimits.MAX_VALUE_OF_DINT_WHICH_CAN_BE_HELD_IN_A_BYTE;
	actual : BYTE;
	converted : BOOL;
	equal : BOOL;
END_VAR
TEST('Check_DINT_TO_BYTE_Max');

// @TEST-RUN
converted := TryConvert_DINT_TO_Destination(value, actual);
equal := actual = DINT_TO_BYTE(value);

// @TEST-ASSERT
AssertTrue(Condition := equal, Message := 'Did not convert DINT to BYTE correctly');
AssertTrue(Condition := converted, Message := 'Did not report DINT to BYTE conversion was successful');

TEST_FINISHED();
END_METHOD

METHOD PUBLIC Check_DINT_TO_BYTE_Min
VAR
	value : DINT := DatatypeLimits.MIN_VALUE_OF_DINT_WHICH_CAN_BE_HELD_IN_A_BYTE;
	actual : BYTE;
	converted : BOOL;
	equal : BOOL;
END_VAR
TEST('Check_DINT_TO_BYTE_Min');

// @TEST-RUN
converted := TryConvert_DINT_TO_Destination(value, actual);
equal := actual = DINT_TO_BYTE(value);

// @TEST-ASSERT
AssertTrue(Condition := equal, Message := 'Did not convert DINT to BYTE correctly');
AssertTrue(Condition := converted, Message := 'Did not report DINT to BYTE conversion was successful');

TEST_FINISHED();
END_METHOD

METHOD PUBLIC Check_DINT_TO_BYTE_TooHigh
VAR
	value : DINT := DatatypeLimits.DINT_MAX_VALUE;
	actual : BYTE;
	converted : BOOL;
END_VAR
TEST('Check_DINT_TO_BYTE_TooHigh');

// @TEST-RUN
converted := TryConvert_DINT_TO_Destination(value, actual);

// @TEST-ASSERT
AssertFalse(Condition := converted, Message := 'Did not report DINT to BYTE conversion was prevented');

TEST_FINISHED();
END_METHOD

METHOD PUBLIC Check_DINT_TO_BYTE_TooLow
VAR
	value : DINT := DatatypeLimits.DINT_MIN_VALUE;
	actual : BYTE;
	converted : BOOL;
END_VAR
TEST('Check_DINT_TO_BYTE_TooLow');

// @TEST-RUN
converted := TryConvert_DINT_TO_Destination(value, actual);

// @TEST-ASSERT
AssertFalse(Condition := converted, Message := 'Did not report DINT to BYTE conversion was prevented');

TEST_FINISHED();
END_METHOD

METHOD PUBLIC Check_DINT_TO_DATE_Max
VAR
	value : DINT := DatatypeLimits.DINT_MAX_VALUE;
	actual : DATE;
	converted : BOOL;
	equal : BOOL;
END_VAR
TEST('Check_DINT_TO_DATE_Max');

// @TEST-RUN
converted := TryConvert_DINT_TO_Destination(value, actual);
equal := actual = DINT_TO_DATE(value);

// @TEST-ASSERT
AssertTrue(Condition := equal, Message := 'Did not convert DINT to DATE correctly');
AssertTrue(Condition := converted, Message := 'Did not report DINT to DATE conversion was successful');

TEST_FINISHED();
END_METHOD

METHOD PUBLIC Check_DINT_TO_DATE_Min
VAR
	value : DINT := DatatypeLimits.MIN_VALUE_OF_DINT_WHICH_CAN_BE_HELD_IN_A_DATE;
	actual : DATE;
	converted : BOOL;
	equal : BOOL;
END_VAR
TEST('Check_DINT_TO_DATE_Min');

// @TEST-RUN
converted := TryConvert_DINT_TO_Destination(value, actual);
equal := actual = DINT_TO_DATE(value);

// @TEST-ASSERT
AssertTrue(Condition := equal, Message := 'Did not convert DINT to DATE correctly');
AssertTrue(Condition := converted, Message := 'Did not report DINT to DATE conversion was successful');

TEST_FINISHED();
END_METHOD

METHOD PUBLIC Check_DINT_TO_DATE_TooLow
VAR
	value : DINT := DatatypeLimits.DINT_MIN_VALUE;
	actual : DATE;
	converted : BOOL;
END_VAR
TEST('Check_DINT_TO_DATE_TooLow');

// @TEST-RUN
converted := TryConvert_DINT_TO_Destination(value, actual);

// @TEST-ASSERT
AssertFalse(Condition := converted, Message := 'Did not report DINT to DATE conversion was prevented');

TEST_FINISHED();
END_METHOD

METHOD PUBLIC Check_DINT_TO_DINT_Max
VAR
	value : DINT := DatatypeLimits.DINT_MAX_VALUE;
	actual : DINT;
	converted : BOOL;
	equal : BOOL;
END_VAR
TEST('Check_DINT_TO_DINT_Max');

// @TEST-RUN
converted := TryConvert_DINT_TO_Destination(value, actual);
equal := actual = value;

// @TEST-ASSERT
AssertTrue(Condition := equal, Message := 'Did not convert DINT to DINT correctly');
AssertTrue(Condition := converted, Message := 'Did not report DINT to DINT conversion was successful');

TEST_FINISHED();
END_METHOD

METHOD PUBLIC Check_DINT_TO_DINT_Min
VAR
	value : DINT := DatatypeLimits.DINT_MIN_VALUE;
	actual : DINT;
	converted : BOOL;
	equal : BOOL;
END_VAR
TEST('Check_DINT_TO_DINT_Min');

// @TEST-RUN
converted := TryConvert_DINT_TO_Destination(value, actual);
equal := actual = value;

// @TEST-ASSERT
AssertTrue(Condition := equal, Message := 'Did not convert DINT to DINT correctly');
AssertTrue(Condition := converted, Message := 'Did not report DINT to DINT conversion was successful');

TEST_FINISHED();
END_METHOD

METHOD PUBLIC Check_DINT_TO_DT_Max
VAR
	value : DINT := DatatypeLimits.DINT_MAX_VALUE;
	actual : DT;
	converted : BOOL;
	equal : BOOL;
END_VAR
TEST('Check_DINT_TO_DT_Max');

// @TEST-RUN
converted := TryConvert_DINT_TO_Destination(value, actual);
equal := actual = DINT_TO_DT(value);

// @TEST-ASSERT
AssertTrue(Condition := equal, Message := 'Did not convert DINT to DT correctly');
AssertTrue(Condition := converted, Message := 'Did not report DINT to DT conversion was successful');

TEST_FINISHED();
END_METHOD

METHOD PUBLIC Check_DINT_TO_DT_Min
VAR
	value : DINT := DatatypeLimits.MIN_VALUE_OF_DINT_WHICH_CAN_BE_HELD_IN_A_DT;
	actual : DT;
	converted : BOOL;
	equal : BOOL;
END_VAR
TEST('Check_DINT_TO_DT_Min');

// @TEST-RUN
converted := TryConvert_DINT_TO_Destination(value, actual);
equal := actual = DINT_TO_DT(value);

// @TEST-ASSERT
AssertTrue(Condition := equal, Message := 'Did not convert DINT to DT correctly');
AssertTrue(Condition := converted, Message := 'Did not report DINT to DT conversion was successful');

TEST_FINISHED();
END_METHOD

METHOD PUBLIC Check_DINT_TO_DT_TooLow
VAR
	value : DINT := DatatypeLimits.DINT_MIN_VALUE;
	actual : DT;
	converted : BOOL;
END_VAR
TEST('Check_DINT_TO_DT_TooLow');

// @TEST-RUN
converted := TryConvert_DINT_TO_Destination(value, actual);

// @TEST-ASSERT
AssertFalse(Condition := converted, Message := 'Did not report DINT to DT conversion was prevented');

TEST_FINISHED();
END_METHOD

METHOD PUBLIC Check_DINT_TO_DWORD_Max
VAR
	value : DINT := DatatypeLimits.DINT_MAX_VALUE;
	actual : DWORD;
	converted : BOOL;
	equal : BOOL;
END_VAR
TEST('Check_DINT_TO_DWORD_Max');

// @TEST-RUN
converted := TryConvert_DINT_TO_Destination(value, actual);
equal := actual = DINT_TO_DWORD(value);

// @TEST-ASSERT
AssertTrue(Condition := equal, Message := 'Did not convert DINT to DWORD correctly');
AssertTrue(Condition := converted, Message := 'Did not report DINT to DWORD conversion was successful');

TEST_FINISHED();
END_METHOD

METHOD PUBLIC Check_DINT_TO_DWORD_Min
VAR
	value : DINT := DatatypeLimits.MIN_VALUE_OF_DINT_WHICH_CAN_BE_HELD_IN_A_DWORD;
	actual : DWORD;
	converted : BOOL;
	equal : BOOL;
END_VAR
TEST('Check_DINT_TO_DWORD_Min');

// @TEST-RUN
converted := TryConvert_DINT_TO_Destination(value, actual);
equal := actual = DINT_TO_DWORD(value);

// @TEST-ASSERT
AssertTrue(Condition := equal, Message := 'Did not convert DINT to DWORD correctly');
AssertTrue(Condition := converted, Message := 'Did not report DINT to DWORD conversion was successful');

TEST_FINISHED();
END_METHOD

METHOD PUBLIC Check_DINT_TO_DWORD_TooLow
VAR
	value : DINT := DatatypeLimits.DINT_MIN_VALUE;
	actual : DWORD;
	converted : BOOL;
END_VAR
TEST('Check_DINT_TO_DWORD_TooLow');

// @TEST-RUN
converted := TryConvert_DINT_TO_Destination(value, actual);

// @TEST-ASSERT
AssertFalse(Condition := converted, Message := 'Did not report DINT to DWORD conversion was prevented');

TEST_FINISHED();
END_METHOD

METHOD PUBLIC Check_DINT_TO_INT_Max
VAR
	value : DINT := DatatypeLimits.MAX_VALUE_OF_DINT_WHICH_CAN_BE_HELD_IN_A_INT;
	actual : INT;
	converted : BOOL;
	equal : BOOL;
END_VAR
TEST('Check_DINT_TO_INT_Max');

// @TEST-RUN
converted := TryConvert_DINT_TO_Destination(value, actual);
equal := actual = DINT_TO_INT(value);

// @TEST-ASSERT
AssertTrue(Condition := equal, Message := 'Did not convert DINT to INT correctly');
AssertTrue(Condition := converted, Message := 'Did not report DINT to INT conversion was successful');

TEST_FINISHED();
END_METHOD

METHOD PUBLIC Check_DINT_TO_INT_Min
VAR
	value : DINT := DatatypeLimits.MIN_VALUE_OF_DINT_WHICH_CAN_BE_HELD_IN_A_INT;
	actual : INT;
	converted : BOOL;
	equal : BOOL;
END_VAR
TEST('Check_DINT_TO_INT_Min');

// @TEST-RUN
converted := TryConvert_DINT_TO_Destination(value, actual);
equal := actual = DINT_TO_INT(value);

// @TEST-ASSERT
AssertTrue(Condition := equal, Message := 'Did not convert DINT to INT correctly');
AssertTrue(Condition := converted, Message := 'Did not report DINT to INT conversion was successful');

TEST_FINISHED();
END_METHOD

METHOD PUBLIC Check_DINT_TO_INT_TooHigh
VAR
	value : DINT := DatatypeLimits.DINT_MAX_VALUE;
	actual : INT;
	converted : BOOL;
END_VAR
TEST('Check_DINT_TO_INT_TooHigh');

// @TEST-RUN
converted := TryConvert_DINT_TO_Destination(value, actual);

// @TEST-ASSERT
AssertFalse(Condition := converted, Message := 'Did not report DINT to INT conversion was prevented');

TEST_FINISHED();
END_METHOD

METHOD PUBLIC Check_DINT_TO_INT_TooLow
VAR
	value : DINT := DatatypeLimits.DINT_MIN_VALUE;
	actual : INT;
	converted : BOOL;
END_VAR
TEST('Check_DINT_TO_INT_TooLow');

// @TEST-RUN
converted := TryConvert_DINT_TO_Destination(value, actual);

// @TEST-ASSERT
AssertFalse(Condition := converted, Message := 'Did not report DINT to INT conversion was prevented');

TEST_FINISHED();
END_METHOD

METHOD PUBLIC Check_DINT_TO_LINT_Max
VAR
	value : DINT := DatatypeLimits.DINT_MAX_VALUE;
	actual : LINT;
	converted : BOOL;
	equal : BOOL;
END_VAR
TEST('Check_DINT_TO_LINT_Max');

// @TEST-RUN
converted := TryConvert_DINT_TO_Destination(value, actual);
equal := actual = DINT_TO_LINT(value);

// @TEST-ASSERT
AssertTrue(Condition := equal, Message := 'Did not convert DINT to LINT correctly');
AssertTrue(Condition := converted, Message := 'Did not report DINT to LINT conversion was successful');

TEST_FINISHED();
END_METHOD

METHOD PUBLIC Check_DINT_TO_LINT_Min
VAR
	value : DINT := DatatypeLimits.DINT_MIN_VALUE;
	actual : LINT;
	converted : BOOL;
	equal : BOOL;
END_VAR
TEST('Check_DINT_TO_LINT_Min');

// @TEST-RUN
converted := TryConvert_DINT_TO_Destination(value, actual);
equal := actual = DINT_TO_LINT(value);

// @TEST-ASSERT
AssertTrue(Condition := equal, Message := 'Did not convert DINT to LINT correctly');
AssertTrue(Condition := converted, Message := 'Did not report DINT to LINT conversion was successful');

TEST_FINISHED();
END_METHOD

METHOD PUBLIC Check_DINT_TO_LREAL_Max
VAR
	value : DINT := DatatypeLimits.DINT_MAX_VALUE;
	actual : LREAL;
	converted : BOOL;
	equal : BOOL;
END_VAR
TEST('Check_DINT_TO_LREAL_Max');

// @TEST-RUN
converted := TryConvert_DINT_TO_Destination(value, actual);
equal := actual = DINT_TO_LREAL(value);

// @TEST-ASSERT
AssertTrue(Condition := equal, Message := 'Did not convert DINT to LREAL correctly');
AssertTrue(Condition := converted, Message := 'Did not report DINT to LREAL conversion was successful');

TEST_FINISHED();
END_METHOD

METHOD PUBLIC Check_DINT_TO_LREAL_Min
VAR
	value : DINT := DatatypeLimits.DINT_MIN_VALUE;
	actual : LREAL;
	converted : BOOL;
	equal : BOOL;
END_VAR
TEST('Check_DINT_TO_LREAL_Min');

// @TEST-RUN
converted := TryConvert_DINT_TO_Destination(value, actual);
equal := actual = DINT_TO_LREAL(value);

// @TEST-ASSERT
AssertTrue(Condition := equal, Message := 'Did not convert DINT to LREAL correctly');
AssertTrue(Condition := converted, Message := 'Did not report DINT to LREAL conversion was successful');

TEST_FINISHED();
END_METHOD

METHOD PUBLIC Check_DINT_TO_LWORD_Max
VAR
	value : DINT := DatatypeLimits.DINT_MAX_VALUE;
	actual : LWORD;
	converted : BOOL;
	equal : BOOL;
END_VAR
TEST('Check_DINT_TO_LWORD_Max');

// @TEST-RUN
converted := TryConvert_DINT_TO_Destination(value, actual);
equal := actual = DINT_TO_LWORD(value);

// @TEST-ASSERT
AssertTrue(Condition := equal, Message := 'Did not convert DINT to LWORD correctly');
AssertTrue(Condition := converted, Message := 'Did not report DINT to LWORD conversion was successful');

TEST_FINISHED();
END_METHOD

METHOD PUBLIC Check_DINT_TO_LWORD_Min
VAR
	value : DINT := DatatypeLimits.MIN_VALUE_OF_DINT_WHICH_CAN_BE_HELD_IN_A_LWORD;
	actual : LWORD;
	converted : BOOL;
	equal : BOOL;
END_VAR
TEST('Check_DINT_TO_LWORD_Min');

// @TEST-RUN
converted := TryConvert_DINT_TO_Destination(value, actual);
equal := actual = DINT_TO_LWORD(value);

// @TEST-ASSERT
AssertTrue(Condition := equal, Message := 'Did not convert DINT to LWORD correctly');
AssertTrue(Condition := converted, Message := 'Did not report DINT to LWORD conversion was successful');

TEST_FINISHED();
END_METHOD

METHOD PUBLIC Check_DINT_TO_LWORD_TooLow
VAR
	value : DINT := DatatypeLimits.DINT_MIN_VALUE;
	actual : LWORD;
	converted : BOOL;
END_VAR
TEST('Check_DINT_TO_LWORD_TooLow');

// @TEST-RUN
converted := TryConvert_DINT_TO_Destination(value, actual);

// @TEST-ASSERT
AssertFalse(Condition := converted, Message := 'Did not report DINT to LWORD conversion was prevented');

TEST_FINISHED();
END_METHOD

METHOD PUBLIC Check_DINT_TO_REAL_Max
VAR
	value : DINT := DatatypeLimits.DINT_MAX_VALUE;
	actual : REAL;
	converted : BOOL;
	equal : BOOL;
END_VAR
TEST('Check_DINT_TO_REAL_Max');

// @TEST-RUN
converted := TryConvert_DINT_TO_Destination(value, actual);
equal := actual = DINT_TO_REAL(value);

// @TEST-ASSERT
AssertTrue(Condition := equal, Message := 'Did not convert DINT to REAL correctly');
AssertTrue(Condition := converted, Message := 'Did not report DINT to REAL conversion was successful');

TEST_FINISHED();
END_METHOD

METHOD PUBLIC Check_DINT_TO_REAL_Min
VAR
	value : DINT := DatatypeLimits.DINT_MIN_VALUE;
	actual : REAL;
	converted : BOOL;
	equal : BOOL;
END_VAR
TEST('Check_DINT_TO_REAL_Min');

// @TEST-RUN
converted := TryConvert_DINT_TO_Destination(value, actual);
equal := actual = DINT_TO_REAL(value);

// @TEST-ASSERT
AssertTrue(Condition := equal, Message := 'Did not convert DINT to REAL correctly');
AssertTrue(Condition := converted, Message := 'Did not report DINT to REAL conversion was successful');

TEST_FINISHED();
END_METHOD

METHOD PUBLIC Check_DINT_TO_SINT_Max
VAR
	value : DINT := DatatypeLimits.MAX_VALUE_OF_DINT_WHICH_CAN_BE_HELD_IN_A_SINT;
	actual : SINT;
	converted : BOOL;
	equal : BOOL;
END_VAR
TEST('Check_DINT_TO_SINT_Max');

// @TEST-RUN
converted := TryConvert_DINT_TO_Destination(value, actual);
equal := actual = DINT_TO_SINT(value);

// @TEST-ASSERT
AssertTrue(Condition := equal, Message := 'Did not convert DINT to SINT correctly');
AssertTrue(Condition := converted, Message := 'Did not report DINT to SINT conversion was successful');

TEST_FINISHED();
END_METHOD

METHOD PUBLIC Check_DINT_TO_SINT_Min
VAR
	value : DINT := DatatypeLimits.MIN_VALUE_OF_DINT_WHICH_CAN_BE_HELD_IN_A_SINT;
	actual : SINT;
	converted : BOOL;
	equal : BOOL;
END_VAR
TEST('Check_DINT_TO_SINT_Min');

// @TEST-RUN
converted := TryConvert_DINT_TO_Destination(value, actual);
equal := actual = DINT_TO_SINT(value);

// @TEST-ASSERT
AssertTrue(Condition := equal, Message := 'Did not convert DINT to SINT correctly');
AssertTrue(Condition := converted, Message := 'Did not report DINT to SINT conversion was successful');

TEST_FINISHED();
END_METHOD

METHOD PUBLIC Check_DINT_TO_SINT_TooHigh
VAR
	value : DINT := DatatypeLimits.DINT_MAX_VALUE;
	actual : SINT;
	converted : BOOL;
END_VAR
TEST('Check_DINT_TO_SINT_TooHigh');

// @TEST-RUN
converted := TryConvert_DINT_TO_Destination(value, actual);

// @TEST-ASSERT
AssertFalse(Condition := converted, Message := 'Did not report DINT to SINT conversion was prevented');

TEST_FINISHED();
END_METHOD

METHOD PUBLIC Check_DINT_TO_SINT_TooLow
VAR
	value : DINT := DatatypeLimits.DINT_MIN_VALUE;
	actual : SINT;
	converted : BOOL;
END_VAR
TEST('Check_DINT_TO_SINT_TooLow');

// @TEST-RUN
converted := TryConvert_DINT_TO_Destination(value, actual);

// @TEST-ASSERT
AssertFalse(Condition := converted, Message := 'Did not report DINT to SINT conversion was prevented');

TEST_FINISHED();
END_METHOD

METHOD PUBLIC Check_DINT_TO_STRING_Max
VAR
	value : DINT := DatatypeLimits.DINT_MAX_VALUE;
	actual : STRING;
	converted : BOOL;
	equal : BOOL;
END_VAR
TEST('Check_DINT_TO_STRING_Max');

// @TEST-RUN
converted := TryConvert_DINT_TO_Destination(value, actual);
equal := actual = DINT_TO_STRING(value);

// @TEST-ASSERT
AssertTrue(Condition := equal, Message := 'Did not convert DINT to STRING correctly');
AssertTrue(Condition := converted, Message := 'Did not report DINT to STRING conversion was successful');

TEST_FINISHED();
END_METHOD

METHOD PUBLIC Check_DINT_TO_STRING_Min
VAR
	value : DINT := DatatypeLimits.DINT_MIN_VALUE;
	actual : STRING;
	converted : BOOL;
	equal : BOOL;
END_VAR
TEST('Check_DINT_TO_STRING_Min');

// @TEST-RUN
converted := TryConvert_DINT_TO_Destination(value, actual);
equal := actual = DINT_TO_STRING(value);

// @TEST-ASSERT
AssertTrue(Condition := equal, Message := 'Did not convert DINT to STRING correctly');
AssertTrue(Condition := converted, Message := 'Did not report DINT to STRING conversion was successful');

TEST_FINISHED();
END_METHOD

METHOD PUBLIC Check_DINT_TO_TIME_Max
VAR
	value : DINT := DatatypeLimits.DINT_MAX_VALUE;
	actual : TIME;
	converted : BOOL;
	equal : BOOL;
END_VAR
TEST('Check_DINT_TO_TIME_Max');

// @TEST-RUN
converted := TryConvert_DINT_TO_Destination(value, actual);
equal := actual = DINT_TO_TIME(value);

// @TEST-ASSERT
AssertTrue(Condition := equal, Message := 'Did not convert DINT to TIME correctly');
AssertTrue(Condition := converted, Message := 'Did not report DINT to TIME conversion was successful');

TEST_FINISHED();
END_METHOD

METHOD PUBLIC Check_DINT_TO_TIME_Min
VAR
	value : DINT := DatatypeLimits.MIN_VALUE_OF_DINT_WHICH_CAN_BE_HELD_IN_A_TIME;
	actual : TIME;
	converted : BOOL;
	equal : BOOL;
END_VAR
TEST('Check_DINT_TO_TIME_Min');

// @TEST-RUN
converted := TryConvert_DINT_TO_Destination(value, actual);
equal := actual = DINT_TO_TIME(value);

// @TEST-ASSERT
AssertTrue(Condition := equal, Message := 'Did not convert DINT to TIME correctly');
AssertTrue(Condition := converted, Message := 'Did not report DINT to TIME conversion was successful');

TEST_FINISHED();
END_METHOD

METHOD PUBLIC Check_DINT_TO_TIME_TooLow
VAR
	value : DINT := DatatypeLimits.DINT_MIN_VALUE;
	actual : TIME;
	converted : BOOL;
END_VAR
TEST('Check_DINT_TO_TIME_TooLow');

// @TEST-RUN
converted := TryConvert_DINT_TO_Destination(value, actual);

// @TEST-ASSERT
AssertFalse(Condition := converted, Message := 'Did not report DINT to TIME conversion was prevented');

TEST_FINISHED();
END_METHOD

METHOD PUBLIC Check_DINT_TO_TOD_Max
VAR
	value : DINT := DatatypeLimits.MAX_VALUE_OF_DINT_WHICH_CAN_BE_HELD_IN_A_TOD;
	actual : TOD;
	converted : BOOL;
	equal : BOOL;
END_VAR
TEST('Check_DINT_TO_TOD_Max');

// @TEST-RUN
converted := TryConvert_DINT_TO_Destination(value, actual);
equal := actual = DINT_TO_TOD(value);

// @TEST-ASSERT
AssertTrue(Condition := equal, Message := 'Did not convert DINT to TOD correctly');
AssertTrue(Condition := converted, Message := 'Did not report DINT to TOD conversion was successful');

TEST_FINISHED();
END_METHOD

METHOD PUBLIC Check_DINT_TO_TOD_Min
VAR
	value : DINT := DatatypeLimits.MIN_VALUE_OF_DINT_WHICH_CAN_BE_HELD_IN_A_TOD;
	actual : TOD;
	converted : BOOL;
	equal : BOOL;
END_VAR
TEST('Check_DINT_TO_TOD_Min');

// @TEST-RUN
converted := TryConvert_DINT_TO_Destination(value, actual);
equal := actual = DINT_TO_TOD(value);

// @TEST-ASSERT
AssertTrue(Condition := equal, Message := 'Did not convert DINT to TOD correctly');
AssertTrue(Condition := converted, Message := 'Did not report DINT to TOD conversion was successful');

TEST_FINISHED();
END_METHOD

METHOD PUBLIC Check_DINT_TO_TOD_TooHigh
VAR
	value : DINT := DatatypeLimits.DINT_MAX_VALUE;
	actual : TOD;
	converted : BOOL;
END_VAR
TEST('Check_DINT_TO_TOD_TooHigh');

// @TEST-RUN
converted := TryConvert_DINT_TO_Destination(value, actual);

// @TEST-ASSERT
AssertFalse(Condition := converted, Message := 'Did not report DINT to TOD conversion was prevented');

TEST_FINISHED();
END_METHOD

METHOD PUBLIC Check_DINT_TO_TOD_TooLow
VAR
	value : DINT := DatatypeLimits.DINT_MIN_VALUE;
	actual : TOD;
	converted : BOOL;
END_VAR
TEST('Check_DINT_TO_TOD_TooLow');

// @TEST-RUN
converted := TryConvert_DINT_TO_Destination(value, actual);

// @TEST-ASSERT
AssertFalse(Condition := converted, Message := 'Did not report DINT to TOD conversion was prevented');

TEST_FINISHED();
END_METHOD

METHOD PUBLIC Check_DINT_TO_UDINT_Max
VAR
	value : DINT := DatatypeLimits.DINT_MAX_VALUE;
	actual : UDINT;
	converted : BOOL;
	equal : BOOL;
END_VAR
TEST('Check_DINT_TO_UDINT_Max');

// @TEST-RUN
converted := TryConvert_DINT_TO_Destination(value, actual);
equal := actual = DINT_TO_UDINT(value);

// @TEST-ASSERT
AssertTrue(Condition := equal, Message := 'Did not convert DINT to UDINT correctly');
AssertTrue(Condition := converted, Message := 'Did not report DINT to UDINT conversion was successful');

TEST_FINISHED();
END_METHOD

METHOD PUBLIC Check_DINT_TO_UDINT_Min
VAR
	value : DINT := DatatypeLimits.MIN_VALUE_OF_DINT_WHICH_CAN_BE_HELD_IN_A_UDINT;
	actual : UDINT;
	converted : BOOL;
	equal : BOOL;
END_VAR
TEST('Check_DINT_TO_UDINT_Min');

// @TEST-RUN
converted := TryConvert_DINT_TO_Destination(value, actual);
equal := actual = DINT_TO_UDINT(value);

// @TEST-ASSERT
AssertTrue(Condition := equal, Message := 'Did not convert DINT to UDINT correctly');
AssertTrue(Condition := converted, Message := 'Did not report DINT to UDINT conversion was successful');

TEST_FINISHED();
END_METHOD

METHOD PUBLIC Check_DINT_TO_UDINT_TooLow
VAR
	value : DINT := DatatypeLimits.DINT_MIN_VALUE;
	actual : UDINT;
	converted : BOOL;
END_VAR
TEST('Check_DINT_TO_UDINT_TooLow');

// @TEST-RUN
converted := TryConvert_DINT_TO_Destination(value, actual);

// @TEST-ASSERT
AssertFalse(Condition := converted, Message := 'Did not report DINT to UDINT conversion was prevented');

TEST_FINISHED();
END_METHOD

METHOD PUBLIC Check_DINT_TO_UINT_Max
VAR
	value : DINT := DatatypeLimits.MAX_VALUE_OF_DINT_WHICH_CAN_BE_HELD_IN_A_UINT;
	actual : UINT;
	converted : BOOL;
	equal : BOOL;
END_VAR
TEST('Check_DINT_TO_UINT_Max');

// @TEST-RUN
converted := TryConvert_DINT_TO_Destination(value, actual);
equal := actual = DINT_TO_UINT(value);

// @TEST-ASSERT
AssertTrue(Condition := equal, Message := 'Did not convert DINT to UINT correctly');
AssertTrue(Condition := converted, Message := 'Did not report DINT to UINT conversion was successful');

TEST_FINISHED();
END_METHOD

METHOD PUBLIC Check_DINT_TO_UINT_Min
VAR
	value : DINT := DatatypeLimits.MIN_VALUE_OF_DINT_WHICH_CAN_BE_HELD_IN_A_UINT;
	actual : UINT;
	converted : BOOL;
	equal : BOOL;
END_VAR
TEST('Check_DINT_TO_UINT_Min');

// @TEST-RUN
converted := TryConvert_DINT_TO_Destination(value, actual);
equal := actual = DINT_TO_UINT(value);

// @TEST-ASSERT
AssertTrue(Condition := equal, Message := 'Did not convert DINT to UINT correctly');
AssertTrue(Condition := converted, Message := 'Did not report DINT to UINT conversion was successful');

TEST_FINISHED();
END_METHOD

METHOD PUBLIC Check_DINT_TO_UINT_TooHigh
VAR
	value : DINT := DatatypeLimits.DINT_MAX_VALUE;
	actual : UINT;
	converted : BOOL;
END_VAR
TEST('Check_DINT_TO_UINT_TooHigh');

// @TEST-RUN
converted := TryConvert_DINT_TO_Destination(value, actual);

// @TEST-ASSERT
AssertFalse(Condition := converted, Message := 'Did not report DINT to UINT conversion was prevented');

TEST_FINISHED();
END_METHOD

METHOD PUBLIC Check_DINT_TO_UINT_TooLow
VAR
	value : DINT := DatatypeLimits.DINT_MIN_VALUE;
	actual : UINT;
	converted : BOOL;
END_VAR
TEST('Check_DINT_TO_UINT_TooLow');

// @TEST-RUN
converted := TryConvert_DINT_TO_Destination(value, actual);

// @TEST-ASSERT
AssertFalse(Condition := converted, Message := 'Did not report DINT to UINT conversion was prevented');

TEST_FINISHED();
END_METHOD

METHOD PUBLIC Check_DINT_TO_ULINT_Max
VAR
	value : DINT := DatatypeLimits.DINT_MAX_VALUE;
	actual : ULINT;
	converted : BOOL;
	equal : BOOL;
END_VAR
TEST('Check_DINT_TO_ULINT_Max');

// @TEST-RUN
converted := TryConvert_DINT_TO_Destination(value, actual);
equal := actual = DINT_TO_ULINT(value);

// @TEST-ASSERT
AssertTrue(Condition := equal, Message := 'Did not convert DINT to ULINT correctly');
AssertTrue(Condition := converted, Message := 'Did not report DINT to ULINT conversion was successful');

TEST_FINISHED();
END_METHOD

METHOD PUBLIC Check_DINT_TO_ULINT_Min
VAR
	value : DINT := DatatypeLimits.MIN_VALUE_OF_DINT_WHICH_CAN_BE_HELD_IN_A_ULINT;
	actual : ULINT;
	converted : BOOL;
	equal : BOOL;
END_VAR
TEST('Check_DINT_TO_ULINT_Min');

// @TEST-RUN
converted := TryConvert_DINT_TO_Destination(value, actual);
equal := actual = DINT_TO_ULINT(value);

// @TEST-ASSERT
AssertTrue(Condition := equal, Message := 'Did not convert DINT to ULINT correctly');
AssertTrue(Condition := converted, Message := 'Did not report DINT to ULINT conversion was successful');

TEST_FINISHED();
END_METHOD

METHOD PUBLIC Check_DINT_TO_ULINT_TooLow
VAR
	value : DINT := DatatypeLimits.DINT_MIN_VALUE;
	actual : ULINT;
	converted : BOOL;
END_VAR
TEST('Check_DINT_TO_ULINT_TooLow');

// @TEST-RUN
converted := TryConvert_DINT_TO_Destination(value, actual);

// @TEST-ASSERT
AssertFalse(Condition := converted, Message := 'Did not report DINT to ULINT conversion was prevented');

TEST_FINISHED();
END_METHOD

METHOD PUBLIC Check_DINT_TO_USINT_Max
VAR
	value : DINT := DatatypeLimits.MAX_VALUE_OF_DINT_WHICH_CAN_BE_HELD_IN_A_USINT;
	actual : USINT;
	converted : BOOL;
	equal : BOOL;
END_VAR
TEST('Check_DINT_TO_USINT_Max');

// @TEST-RUN
converted := TryConvert_DINT_TO_Destination(value, actual);
equal := actual = DINT_TO_USINT(value);

// @TEST-ASSERT
AssertTrue(Condition := equal, Message := 'Did not convert DINT to USINT correctly');
AssertTrue(Condition := converted, Message := 'Did not report DINT to USINT conversion was successful');

TEST_FINISHED();
END_METHOD

METHOD PUBLIC Check_DINT_TO_USINT_Min
VAR
	value : DINT := DatatypeLimits.MIN_VALUE_OF_DINT_WHICH_CAN_BE_HELD_IN_A_USINT;
	actual : USINT;
	converted : BOOL;
	equal : BOOL;
END_VAR
TEST('Check_DINT_TO_USINT_Min');

// @TEST-RUN
converted := TryConvert_DINT_TO_Destination(value, actual);
equal := actual = DINT_TO_USINT(value);

// @TEST-ASSERT
AssertTrue(Condition := equal, Message := 'Did not convert DINT to USINT correctly');
AssertTrue(Condition := converted, Message := 'Did not report DINT to USINT conversion was successful');

TEST_FINISHED();
END_METHOD

METHOD PUBLIC Check_DINT_TO_USINT_TooHigh
VAR
	value : DINT := DatatypeLimits.DINT_MAX_VALUE;
	actual : USINT;
	converted : BOOL;
END_VAR
TEST('Check_DINT_TO_USINT_TooHigh');

// @TEST-RUN
converted := TryConvert_DINT_TO_Destination(value, actual);

// @TEST-ASSERT
AssertFalse(Condition := converted, Message := 'Did not report DINT to USINT conversion was prevented');

TEST_FINISHED();
END_METHOD

METHOD PUBLIC Check_DINT_TO_USINT_TooLow
VAR
	value : DINT := DatatypeLimits.DINT_MIN_VALUE;
	actual : USINT;
	converted : BOOL;
END_VAR
TEST('Check_DINT_TO_USINT_TooLow');

// @TEST-RUN
converted := TryConvert_DINT_TO_Destination(value, actual);

// @TEST-ASSERT
AssertFalse(Condition := converted, Message := 'Did not report DINT to USINT conversion was prevented');

TEST_FINISHED();
END_METHOD

METHOD PUBLIC Check_DINT_TO_WORD_Max
VAR
	value : DINT := DatatypeLimits.MAX_VALUE_OF_DINT_WHICH_CAN_BE_HELD_IN_A_WORD;
	actual : WORD;
	converted : BOOL;
	equal : BOOL;
END_VAR
TEST('Check_DINT_TO_WORD_Max');

// @TEST-RUN
converted := TryConvert_DINT_TO_Destination(value, actual);
equal := actual = DINT_TO_WORD(value);

// @TEST-ASSERT
AssertTrue(Condition := equal, Message := 'Did not convert DINT to WORD correctly');
AssertTrue(Condition := converted, Message := 'Did not report DINT to WORD conversion was successful');

TEST_FINISHED();
END_METHOD

METHOD PUBLIC Check_DINT_TO_WORD_Min
VAR
	value : DINT := DatatypeLimits.MIN_VALUE_OF_DINT_WHICH_CAN_BE_HELD_IN_A_WORD;
	actual : WORD;
	converted : BOOL;
	equal : BOOL;
END_VAR
TEST('Check_DINT_TO_WORD_Min');

// @TEST-RUN
converted := TryConvert_DINT_TO_Destination(value, actual);
equal := actual = DINT_TO_WORD(value);

// @TEST-ASSERT
AssertTrue(Condition := equal, Message := 'Did not convert DINT to WORD correctly');
AssertTrue(Condition := converted, Message := 'Did not report DINT to WORD conversion was successful');

TEST_FINISHED();
END_METHOD

METHOD PUBLIC Check_DINT_TO_WORD_TooHigh
VAR
	value : DINT := DatatypeLimits.DINT_MAX_VALUE;
	actual : WORD;
	converted : BOOL;
END_VAR
TEST('Check_DINT_TO_WORD_TooHigh');

// @TEST-RUN
converted := TryConvert_DINT_TO_Destination(value, actual);

// @TEST-ASSERT
AssertFalse(Condition := converted, Message := 'Did not report DINT to WORD conversion was prevented');

TEST_FINISHED();
END_METHOD

METHOD PUBLIC Check_DINT_TO_WORD_TooLow
VAR
	value : DINT := DatatypeLimits.DINT_MIN_VALUE;
	actual : WORD;
	converted : BOOL;
END_VAR
TEST('Check_DINT_TO_WORD_TooLow');

// @TEST-RUN
converted := TryConvert_DINT_TO_Destination(value, actual);

// @TEST-ASSERT
AssertFalse(Condition := converted, Message := 'Did not report DINT to WORD conversion was prevented');

TEST_FINISHED();
END_METHOD

END_FUNCTION_BLOCK

// ---- mobject-converters/Tests/INT_TO_TestSuite.TcPOU
FUNCTION_BLOCK PUBLIC INT_TO_TestSuite EXTENDS TcUnit.FB_TestSuite
VAR
END_VAR

Check_INT_TO_BOOL_Max();
Check_INT_TO_BOOL_Min();
Check_INT_TO_BYTE_Max();
Check_INT_TO_BYTE_Min();
Check_INT_TO_BYTE_TooHigh();
Check_INT_TO_BYTE_TooLow();
Check_INT_TO_WORD_Max();
Check_INT_TO_WORD_Min();
Check_INT_TO_WORD_TooLow();
Check_INT_TO_DWORD_Max();
Check_INT_TO_DWORD_Min();
Check_INT_TO_DWORD_TooLow();
Check_INT_TO_LWORD_Max();
Check_INT_TO_LWORD_Min();
Check_INT_TO_LWORD_TooLow();
Check_INT_TO_SINT_Max();
Check_INT_TO_SINT_Min();
Check_INT_TO_SINT_TooHigh();
Check_INT_TO_SINT_TooLow();
Check_INT_TO_INT_Max();
Check_INT_TO_INT_Min();
Check_INT_TO_DINT_Max();
Check_INT_TO_DINT_Min();
Check_INT_TO_LINT_Max();
Check_INT_TO_LINT_Min();
Check_INT_TO_USINT_Max();
Check_INT_TO_USINT_Min();
Check_INT_TO_USINT_TooHigh();
Check_INT_TO_USINT_TooLow();
Check_INT_TO_UINT_Max();
Check_INT_TO_UINT_Min();
Check_INT_TO_UINT_TooLow();
Check_INT_TO_UDINT_Max();
Check_INT_TO_UDINT_Min();
Check_INT_TO_UDINT_TooLow();
Check_INT_TO_ULINT_Max();
Check_INT_TO_ULINT_Min();
Check_INT_TO_ULINT_TooLow();
Check_INT_TO_REAL_Max();
Check_INT_TO_REAL_Min();
Check_INT_TO_LREAL_Max();
Check_INT_TO_LREAL_Min();
Check_INT_TO_TIME_Max();
Check_INT_TO_TIME_Min();
Check_INT_TO_TIME_TooLow();
Check_INT_TO_TOD_Max();
Check_INT_TO_TOD_Min();
Check_INT_TO_TOD_TooLow();
Check_INT_TO_DATE_Max();
Check_INT_TO_DATE_Min();
Check_INT_TO_DATE_TooLow();
Check_INT_TO_DT_Max();
Check_INT_TO_DT_Min();
Check_INT_TO_DT_TooLow();
Check_INT_TO_STRING_Max();
Check_INT_TO_STRING_Min();

METHOD PUBLIC Check_INT_TO_BOOL_Max
VAR
	value : INT := DatatypeLimits.INT_MAX_VALUE;
	actual : BOOL;
	converted : BOOL;
	equal : BOOL;
END_VAR
TEST('Check_INT_TO_BOOL_Max');

// @TEST-RUN
converted := TryConvert_INT_TO_Destination(value, actual);
equal := actual = INT_TO_BOOL(value);

// @TEST-ASSERT
AssertTrue(Condition := equal, Message := 'Did not convert INT to BOOL correctly');
AssertTrue(Condition := converted, Message := 'Did not report INT to BOOL conversion was successful');

TEST_FINISHED();
END_METHOD

METHOD PUBLIC Check_INT_TO_BOOL_Min
VAR
	value : INT := DatatypeLimits.INT_MIN_VALUE;
	actual : BOOL;
	converted : BOOL;
	equal : BOOL;
END_VAR
TEST('Check_INT_TO_BOOL_Min');

// @TEST-RUN
converted := TryConvert_INT_TO_Destination(value, actual);
equal := actual = INT_TO_BOOL(value);

// @TEST-ASSERT
AssertTrue(Condition := equal, Message := 'Did not convert INT to BOOL correctly');
AssertTrue(Condition := converted, Message := 'Did not report INT to BOOL conversion was successful');

TEST_FINISHED();
END_METHOD

METHOD PUBLIC Check_INT_TO_BYTE_Max
VAR
	value : INT := DatatypeLimits.MAX_VALUE_OF_INT_WHICH_CAN_BE_HELD_IN_A_BYTE;
	actual : BYTE;
	converted : BOOL;
	equal : BOOL;
END_VAR
TEST('Check_INT_TO_BYTE_Max');

// @TEST-RUN
converted := TryConvert_INT_TO_Destination(value, actual);
equal := actual = INT_TO_BYTE(value);

// @TEST-ASSERT
AssertTrue(Condition := equal, Message := 'Did not convert INT to BYTE correctly');
AssertTrue(Condition := converted, Message := 'Did not report INT to BYTE conversion was successful');

TEST_FINISHED();
END_METHOD

METHOD PUBLIC Check_INT_TO_BYTE_Min
VAR
	value : INT := DatatypeLimits.MIN_VALUE_OF_INT_WHICH_CAN_BE_HELD_IN_A_BYTE;
	actual : BYTE;
	converted : BOOL;
	equal : BOOL;
END_VAR
TEST('Check_INT_TO_BYTE_Min');

// @TEST-RUN
converted := TryConvert_INT_TO_Destination(value, actual);
equal := actual = INT_TO_BYTE(value);

// @TEST-ASSERT
AssertTrue(Condition := equal, Message := 'Did not convert INT to BYTE correctly');
AssertTrue(Condition := converted, Message := 'Did not report INT to BYTE conversion was successful');

TEST_FINISHED();
END_METHOD

METHOD PUBLIC Check_INT_TO_BYTE_TooHigh
VAR
	value : INT := DatatypeLimits.INT_MAX_VALUE;
	actual : BYTE;
	converted : BOOL;
END_VAR
TEST('Check_INT_TO_BYTE_TooHigh');

// @TEST-RUN
converted := TryConvert_INT_TO_Destination(value, actual);

// @TEST-ASSERT
AssertFalse(Condition := converted, Message := 'Did not report INT to BYTE conversion was prevented');

TEST_FINISHED();
END_METHOD

METHOD PUBLIC Check_INT_TO_BYTE_TooLow
VAR
	value : INT := DatatypeLimits.INT_MIN_VALUE;
	actual : BYTE;
	converted : BOOL;
END_VAR
TEST('Check_INT_TO_BYTE_TooLow');

// @TEST-RUN
converted := TryConvert_INT_TO_Destination(value, actual);

